//
CASE stCommand.CoordinateType OF
	DUT_Command_CoordinateType.Literal:
		F_AddElement(_Command, _Delimiter, _CoordTypeH);
		F_AddElement(_Command, _Delimiter, LREAL_TO_STRING(stCommand.CoordRef.X));
		F_AddElement(_Command, _Delimiter, LREAL_TO_STRING(stCommand.CoordRef.Y));
		F_AddElement(_Command, _Delimiter, LREAL_TO_STRING(stCommand.CoordRef.Z));
		F_AddElement(_Command, _Delimiter, LREAL_TO_STRING(stCommand.CoordRef.A));
		F_AddElement(_Command, _Delimiter, LREAL_TO_STRING(stCommand.CoordRef.B));
		F_AddElement(_Command, _Delimiter, LREAL_TO_STRING(stCommand.CoordRef.C));
		
	DUT_Command_CoordinateType.Variable:
		F_AddElement(_Command, _Delimiter, _CoordTypeV);
		CASE stCommand.ArrayType OF
			DUT_Command_ArrayType.StoredPosition:
				F_AddElement(_Command, _Delimiter, _ArrayTypeS);
			DUT_Command_ArrayType.VisionRegister:
				F_AddElement(_Command, _Delimiter, _ArrayTypeV);
			DUT_Command_ArrayType.Flag:
				// on damn
		END_CASE
		F_AddElement(_Command, _Delimiter, UDINT_TO_STRING(stCommand.ArrayIndex));
		
END_CASE

// only add if move type is circle
IF stCommand.MoveType = DUT_Command_MoveType.CircularMove THEN
	//
	CASE stCommand.CircleMode OF
		MC_CIRC_MODE.mcCircModeBorder:
			F_AddElement(_Command, _Delimiter, _CircleModeBor);
		MC_CIRC_MODE.mcCircModeCenter:
			F_AddElement(_Command, _Delimiter, _CircleModeCen);
		MC_CIRC_MODE.mcCircModeRadius:
			F_AddElement(_Command, _Delimiter, _CircleModeRad);
	END_CASE
	//
	CASE stCommand.PathChoice OF
		MC_CIRC_PATHCHOICE.mcCircPathChoiceClockwise:
			F_AddElement(_Command, _Delimiter, _PathChoiceClw);
		MC_CIRC_PATHCHOICE.mcCircPathChoiceCounterClockwise:
			F_AddElement(_Command, _Delimiter, _PathChoiceCcw);
	END_CASE
	//
	CASE stCommand.CircularCoordinateType OF
		DUT_Command_CoordinateType.Literal:
			F_AddElement(_Command, _Delimiter, _CoordTypeH);
			F_AddElement(_Command, _Delimiter, LREAL_TO_STRING(stCommand.CoordRef2.X));
			F_AddElement(_Command, _Delimiter, LREAL_TO_STRING(stCommand.CoordRef2.Y));
			F_AddElement(_Command, _Delimiter, LREAL_TO_STRING(stCommand.CoordRef2.Z));
			F_AddElement(_Command, _Delimiter, LREAL_TO_STRING(stCommand.CoordRef2.A));
			F_AddElement(_Command, _Delimiter, LREAL_TO_STRING(stCommand.CoordRef2.B));
			F_AddElement(_Command, _Delimiter, LREAL_TO_STRING(stCommand.CoordRef2.C));
			
		DUT_Command_CoordinateType.Variable:
			F_AddElement(_Command, _Delimiter, _CoordTypeV);
			CASE stCommand.CircularArrayType OF
				DUT_Command_ArrayType.StoredPosition:
					F_AddElement(_Command, _Delimiter, _ArrayTypeS);
				DUT_Command_ArrayType.VisionRegister:
					F_AddElement(_Command, _Delimiter, _ArrayTypeV);
				DUT_Command_ArrayType.Flag:
					// oh damn
			END_CASE
			F_AddElement(_Command, _Delimiter, UDINT_TO_STRING(stCommand.CircularArrayIndex));
			
	END_CASE

END_IF

// set function equal to command
BuildMoveCmd := _Command;

END_FUNCTION

// ---- FB/F_AddElement.TcPOU
FUNCTION F_AddElement
VAR_IN_OUT
	Command: STRING(GVL.COMMAND_LEN);
END_VAR
VAR_INPUT
	Delimiter: STRING(1):=' '; // default to space
	Element: STRING(GVL.COMMAND_LEN);
END_VAR
VAR
END_VAR

//
// input
// 	Element: 'bar'
// 	Delimiter: ','
// 	Command: 'foo'
//
// output
// 	Command: 'foo,bar'
//

Command:=CONCAT(Command, Element);
Command:=CONCAT(Command, Delimiter);

END_FUNCTION

// ---- FB/home/F_HomeOffsetCalc.TcPOU
FUNCTION F_HomeOffsetCalc : LREAL
VAR_INPUT
	CurrentOffset: LREAL;
	CurrentPosition: LREAL;
	HomeSearchDirection: Tc2_MC2.MC_Direction;
END_VAR

IF (HomeSearchDirection = Tc2_MC2.MC_Direction.MC_Negative_Direction) THEN
	F_HomeOffsetCalc := -F_RoundLreal(ABS(CurrentPosition - CurrentOffset),2);
	
ELSIF (HomeSearchDirection = Tc2_MC2.MC_Direction.MC_Positive_Direction) THEN
	F_HomeOffsetCalc := F_RoundLreal(ABS(CurrentPosition - CurrentOffset),2);
	
ELSE
	F_HomeOffsetCalc := CurrentOffset;
	
END_IF

END_FUNCTION

// ---- FB/F_RoundLreal.TcPOU
FUNCTION F_RoundLreal : LREAL
VAR_INPUT
   rIn : LREAL;      
   Digit: INT;         
END_VAR

VAR
   d1 : DINT;
   r0,r1,r2,Rdigit: LREAL;               
END_VAR

// https://forge.codesys.com/forge/talk/Engineering/thread/8d1ee86294/
rdigit   :=INT_TO_LREAL(Digit);
r0 := EXPT(10,rdigit); 
r1 := rIn * r0;
d1 := TRUNC(r1);
r2 := DINT_TO_LREAL(d1);
F_RoundLreal := r2 / r0;

END_FUNCTION

// ---- FB/jog/FB_JogProcessor.TcPOU
FUNCTION_BLOCK FB_JogProcessor
VAR CONSTANT
	NumberOfAxes: UINT:=GVL.NumberOfAxes;
END_VAR
VAR_IN_OUT
	ACS: ARRAY[1..NumberOfAxes] OF AXIS_REF;
	MCS: ARRAY[1..NumberOfAxes] OF AXIS_REF;
	GroupHandler: FB_GroupHandler;
	//Controller: FB_Controller;
END_VAR
VAR_INPUT
	Enable: BOOL;
	Reset: BOOL;
	Velocity: LREAL := 0;
	Acceleration: LREAL := 0;
	Deceleration: LREAL := 0;
	Jerk: LREAL := 0;
    MaxAngularDistance: LREAL := 90.0;
	MaxLinearDistance: LREAL := 50.0;
// 	AccFactor: LREAL := 1.0;
// 	VelFactor: LREAL := 0.1;
// 	JerkFactor: LREAL := 1.0;
// 	TorqueFactor: LREAL := 1.0;
// 	JogForward: ARRAY[1..NumberOfAxes] OF BOOL;
// 	JogBackwards: ARRAY[1..NumberOfAxes] OF BOOL;
	CoordSystem: DUT_CoordSystem := DUT_CoordSystem.TCP;
	ABC_as_ACS: BOOL;
	StoredPositions: REFERENCE TO ARRAY[GVL.POS_ARR_BEG..GVL.POS_ARR_END] OF DUT_StoredPosition;
	VisionRegisters: REFERENCE TO ARRAY[GVL.VIS_ARR_BEG..GVL.VIS_ARR_END] OF DUT_VisionRegister;
	Flags: REFERENCE TO ARRAY[GVL.FLG_ARR_BEG..GVL.FLG_ARR_END] OF DUT_Flags;
END_VAR
VAR_OUTPUT
	Position: DUT_COORD_REF;
	Enabled: BOOL;
	Done: BOOL;
	Busy: BOOL;
	Error: BOOL;
	ErrorID: UDINT;
END_VAR
VAR
	_ResetRtrig: R_TRIG;
	_ErrorRtrig: R_TRIG;
	_EnableRtrig: R_TRIG;
	_EnableFtrig: F_TRIG;
	
	_SequenceMain: INT;
	_SequenceSetCoordTrans: INT;
	
	_MC_Jog: ARRAY[1..NumberOfAxes*2] OF MC_JOG;
	_MC_Halt: ARRAY[1..NumberOfAxes*2] OF MC_HALT;
	_Halt: ARRAY[1..NumberOfAxes*2] OF BOOL;
	_HaltFtrig: ARRAY[1..NumberOfAxes*2] OF F_Trig;
	_JogForward: ARRAY[1..NumberOfAxes] OF BOOL;
	_JogBackwards: ARRAY[1..NumberOfAxes] OF BOOL;
	_CoordSystem: DUT_CoordSystem := DUT_CoordSystem.TCP;
	
	_ControllerCenter: USINT:=128;
	_ControllerDeadZone: USINT:=40;
	
	_OffsetExist: ARRAY[0..GVL.MCS_POS_IDX-GVL.TCP_POS_IDX] OF BOOL;
	
	_MoveToPose: ARRAY[0..GVL.POSE_5_IDX-GVL.POSE_1_IDX] OF BOOL;
	_MoveCommandProcessor: MoveCmdProcessor;
	
	_i, _j, _k: UINT;
	_FirstScan: BOOL:=TRUE;
	
END_VAR

VAR CONSTANT
	STEP_DONE: 				INT := 1000;
	STEP_IDLE: 				INT := 0000;
	STEP_GROUP_ENABLE: 		INT := 0030;
	STEP_WAIT_ENABLE: 		INT := 0035;
	STEP_SET_KINEMATICS: 	INT := 0060;
	STEP_WAIT_KINEMATICS: 	INT := 0070;
	STEP_JOG:				INT := 0080;
	STEP_WAIT_JOG:			INT := 0090;
	STEP_GROUP_DISABLE: 	INT := 0100;
	STEP_WAIT_DISABLE: 		INT := 0110;
END_VAR

_ResetRtrig(CLK:=Reset);

IF _FirstScan THEN
	//
END_IF

//
_M_HandleController();
_M_HandlePose();

//
_EnableFtrig(CLK:=Enable);
IF _EnableFtrig.Q THEN
	//;
END_IF
_EnableRtrig(CLK:=Enable);
IF _EnableRtrig.Q THEN
	//
END_IF

//
CASE _SequenceMain OF
	STEP_DONE: // done
		Busy := FALSE;
		Done := TRUE;
		_SequenceMain := STEP_IDLE;
		
	STEP_IDLE: // IDLE
		IF _EnableRtrig.Q THEN
			Busy := TRUE;
			Done := FALSE;
			_CoordSystem := CoordSystem;
			_M_CheckOffsets();
			_SequenceMain := STEP_GROUP_ENABLE;
		END_IF
		
	STEP_GROUP_ENABLE:
		IF GroupHandler.M_EnableGroup(_CoordSystem) THEN
			_SequenceMain := STEP_WAIT_ENABLE;
		ELSE
			_SequenceMain := STEP_DONE;
			Error := TRUE;
			ErrorID := GroupHandler.ErrorID;
		END_IF
		
	STEP_WAIT_ENABLE:
		// TODO add timeout timer here
		IF GroupHandler.P_GroupReady THEN
			_SequenceMain := STEP_WAIT_JOG;
		END_IF;
		
	STEP_WAIT_JOG: //
		FOR _k:= 1 TO NumberOfAxes DO
			IF _MC_Jog[_k].Error THEN
				Error := TRUE;
				ErrorID := _MC_Jog[_k].ErrorID;
			END_IF
		END_FOR
		IF _EnableFtrig.Q THEN
			_SequenceMain := STEP_GROUP_DISABLE;
			//_SequenceMain := STEP_DONE;
		END_IF
			
	STEP_GROUP_DISABLE:
		IF GroupHandler.M_DisableGroup() THEN
			_SequenceMain := STEP_WAIT_DISABLE;
		ELSE
			_SequenceMain := STEP_DONE;
			Error := TRUE;
			ErrorID := GroupHandler.ErrorID;
		END_IF
		
	STEP_WAIT_DISABLE:
		// TODO add timeouttimer here
		IF NOT GroupHandler.P_GroupReady THEN
			_SequenceMain := STEP_DONE;
		END_IF
	
END_CASE

//
IF _ResetRtrig.Q AND Error THEN
	Error := FALSE;
	ErrorID := 0;
	_SequenceMain := STEP_DONE;
	GroupHandler.M_ResetGroup();
	_MoveCommandProcessor.M_Home();
END_IF

// https://infosys.beckhoff.com/content/1033/tcplclib_tc2_mc2/70120459.html?id=7121036612998147748
FOR _k:= 1 TO NumberOfAxes DO
	_MC_Jog[_k](
		Axis:= ACS[_k], 
		JogForward:= SEL(_CoordSystem = DUT_CoordSystem.ACS, FALSE, _JogForward[_k]), 
		JogBackwards:= SEL(_CoordSystem = DUT_CoordSystem.ACS, FALSE, _JogBackwards[_k]), 
		Mode:= MC_JOGMODE_INCHING, // MC_JOGMODE_STANDARD_SLOW, MC_JOGMODE_STANDARD_FAST, MC_JOGMODE_CONTINUOUS, MC_JOGMODE_INCHING, MC_JOGMODE_INCHING_MODULO
		Position:= MaxAngularDistance, 
		Velocity:= Velocity, 
		Acceleration:= Acceleration, 
		Deceleration:= Deceleration, 
		Jerk:= Jerk, 
		Done=> , 
		Busy=> , 
		Active=> , 
		CommandAborted=> , 
		Error=> , 
		ErrorID=> );
	_MC_Jog[_k+NumberOfAxes](
		Axis:= MCS[_k], 
		JogForward:= SEL(_CoordSystem = DUT_CoordSystem.MCS, FALSE, _JogForward[_k]), 
		JogBackwards:= SEL(_CoordSystem = DUT_CoordSystem.MCS, FALSE, _JogBackwards[_k]), 
		Mode:= MC_JOGMODE_INCHING, // MC_JOGMODE_STANDARD_SLOW, MC_JOGMODE_STANDARD_FAST, MC_JOGMODE_CONTINUOUS, MC_JOGMODE_INCHING, MC_JOGMODE_INCHING_MODULO
		Position:= MaxLinearDistance, 
		Velocity:= Velocity, 
		Acceleration:= Acceleration, 
		Deceleration:= Deceleration, 
		Jerk:= Jerk, 
		Done=> , 
		Busy=> , 
		Active=> , 
		CommandAborted=> , 
		Error=> , 
		ErrorID=> );
END_FOR
FOR _k:= 1 TO NumberOfAxes DO
	IF _MC_Jog[_k].Error OR _MC_Jog[_k+NumberOfAxes].Error THEN
		//
	END_IF
END_FOR

//
FOR _k:= 1 TO NumberOfAxes DO
	_HaltFtrig[_k](CLK:=_JogForward[_k] OR _JogBackwards[_k]);
	IF _HaltFtrig[_k].Q THEN
		_Halt[_k]:=TRUE;
	END_IF
	_HaltFtrig[_k+NumberOfAxes](CLK:=_JogForward[_k] OR _JogBackwards[_k]);
	IF _HaltFtrig[_k+NumberOfAxes].Q THEN
		_Halt[_k+NumberOfAxes]:=TRUE;
	END_IF
END_FOR
FOR _k:= 1 TO NumberOfAxes DO
	_MC_Halt[_k](
		Axis:= ACS[_k], 
		Execute:= _Halt[_k], 
		Deceleration:= Deceleration, 
		Jerk:= Jerk, 
		BufferMode:= , 
		Options:= , 
		Done=> , 
		Busy=> , 
		Active=> , 
		CommandAborted=> , 
		Error=> , 
		ErrorID=> );
	_MC_Halt[_k+NumberOfAxes](
		Axis:= MCS[_k], 
		Execute:= _Halt[_k+NumberOfAxes], 
		Deceleration:= Deceleration, 
		Jerk:= Jerk, 
		BufferMode:= , 
		Options:= , 
		Done=> , 
		Busy=> , 
		Active=> , 
		CommandAborted=> , 
		Error=> , 
		ErrorID=> );
END_FOR
FOR _k:= 1 TO NumberOfAxes DO
	IF _MC_Halt[_k].Done OR _MC_Halt[_k].Error THEN
		_Halt[_k]:=FALSE;
	END_IF
	IF _MC_Halt[_k+NumberOfAxes].Done OR _MC_Halt[_k+NumberOfAxes].Error THEN
		_Halt[_k+NumberOfAxes]:=FALSE;
	END_IF
END_FOR

//
// CoordSystem := _SMC_GroupJog2.CoordSystem;
// ABC_as_ACS := _SMC_GroupJog2.ABC_as_ACS;
// Enabled := _SMC_GroupJog2.Enable;

//
_ErrorRtrig(CLK:=GroupHandler.Error
				//OR _SMC_GroupJog2.Error
				OR _MoveCommandProcessor.Error);			
IF _ErrorRtrig.Q THEN
	// TODO need to rework how error messages are handled (globally)
	// if the move command processor has an error, we dont know what it is.
	Error := TRUE;
END_IF

// do not put anything after this
_FirstScan := FALSE;

METHOD PRIVATE _M_CheckOffsets : BOOL
VAR
	_i: INT;
	_j: INT;
	_k: INT;
END_VAR
IF Enable THEN
	FOR _j:=0 TO GVL.MCS_POS_IDX-GVL.TCP_POS_IDX BY 1 DO
		_OffsetExist[_j] := FALSE;
	END_FOR
	FOR _i := GVL.TCP_POS_IDX TO GVL.MCS_POS_IDX BY 1 DO
		IF StoredPositions[_i].Position.X <> 0
			OR_ELSE StoredPositions[_i].Position.Y <> 0
			OR_ELSE StoredPositions[_i].Position.Z <> 0
			OR_ELSE StoredPositions[_i].Position.A <> 0
			OR_ELSE StoredPositions[_i].Position.B <> 0
			OR_ELSE StoredPositions[_i].Position.C <> 0 THEN
				_OffsetExist[_i - GVL.TCP_POS_IDX] := TRUE;
		END_IF
	END_FOR
END_IF
END_METHOD

METHOD PRIVATE _M_HandleController : BOOL
VAR_STAT
	OptionsTimer: TON := (PT := TIME#1s0ms);
	OptionsRtrig: R_TRIG;
	ShareTimer: TON := (PT := TIME#1s0ms);
	ShareRtrig: R_TRIG;
	OptionsShareRtrig: R_TRIG;
	JogEnabledRtrig: R_TRIG;
	JogEnabledFtrig: F_TRIG;
	SquareButtonRtrig: R_TRIG;
	TriangleButtonRtrig: R_TRIG;
	CircleButtonRtrig: R_TRIG;
	CrossButtonRtrig: R_TRIG;
	R2_Last: USINT;
	JoyStickLeftXLast: USINT;
	JoyStickLeftYLast: USINT;
	JoyStickRightXLast: USINT;
	JoyStickRightYLast: USINT;
	FactorMin: LREAL := 0.01;
END_VAR
// //
// OptionsTimer(IN:=Controller.P_State.Buttons.Options);
// OptionsRtrig(CLK:=Controller.P_State.Buttons.Options);
// //
// ShareTimer(IN:=Controller.P_State.Buttons.Share);
// ShareRtrig(CLK:=Controller.P_State.Buttons.Share);
// //
// OptionsShareRtrig(CLK:=OptionsTimer.Q AND_THEN ShareTimer.Q);
// JogEnabledRtrig(CLK:=Enable);
// JogEnabledFtrig(CLK:=Enable);
// 
// 
// IF Enable AND_THEN Controller.P_State.Connected THEN
// 	
// 	// toggle jog enable
// 	IF OptionsShareRtrig.Q THEN
// 		//_SMC_GroupJog2.Enable := NOT _SMC_GroupJog2.Enable;
// 	END_IF
// 	IF JogEnabledRtrig.Q OR JogEnabledFtrig.Q THEN
// 		IF Enable THEN
// 			_CoordSystem := DUT_CoordSystem.TCP;
// 			Controller.M_SetTriggerMode(E_ControllerTrigger.Right, E_ControllerTriggerMode.Rigid);
// 			Controller.M_SetTriggerForce(E_ControllerTrigger.Right, E_ControllerTriggerForceParameter.One, 0);
// 			Controller.M_SetPlayerID(E_ControllerPlayerID.PlayerALL);
// 			Controller.M_SetMicrophoneState(TRUE);
// 		ELSE
// 			Controller.M_SetTriggerMode(E_ControllerTrigger.Right, E_ControllerTriggerMode.Off);
// 			Controller.M_SetMicrophoneState(FALSE);
// 		END_IF
// 	END_IF
// 	
// 	// cycle through coord system
// 	IF OptionsRtrig.Q AND NOT Controller.P_State.Buttons.Share THEN
// 		CASE _.CoordSystem OF
// 			DUT_CoordSystem.ACS:
// 				_CoordSystem := DUT_CoordSystem.MCS;
// 				Controller.M_SetPlayerID(E_ControllerPlayerID.Player2);
// 			DUT_CoordSystem.MCS:
// 				_CoordSystem := DUT_CoordSystem.UCS1;
// 				Controller.M_SetPlayerID(E_ControllerPlayerID.Player3);
// 			DUT_CoordSystem.UCS1:
// 				_CoordSystem := DUT_CoordSystem.UCS2;
// 				Controller.M_SetPlayerID(E_ControllerPlayerID.Player4);
// 			DUT_CoordSystem.UCS2:
// 				_CoordSystem := DUT_CoordSystem.TCP;
// 				Controller.M_SetPlayerID(E_ControllerPlayerID.PlayerALL);
// 			DUT_CoordSystem.TCP:
// 				_CoordSystem := DUT_CoordSystem.ACS;
// 				Controller.M_SetPlayerID(E_ControllerPlayerID.Player1);
// // 			DUT_CoordSystem.WCS:
// // 				_CoordSystem := DUT_CoordSystem.ACS;
// // 				Controller.M_SetPlayerID(E_ControllerPlayerID.Player1);
// 		END_CASE
// 	END_IF
// 	
// 	// toggle the ABC as ACS setting
// 	IF ShareRtrig.Q AND NOT Controller.P_State.Buttons.Options THEN
// 		ABC_as_ACS := NOT ABC_as_ACS;
// 	END_IF
// 	
// 	// set the velocity factor while the left trigger button is pressed
// 	IF Controller.P_State.Dpad.Left AND_THEN Controller.P_State.Triggers.Right.Two <> R2_Last THEN
// 		R2_Last := Controller.P_State.Triggers.Right.Two;
// 		//_SMC_GroupJog2.VelFactor := MAX(FactorMin, Controller.P_State.Triggers.Right.Two * 1.0 / 255.0);
// 	END_IF
// 	// set the acceleration factor while the up dpad button is pressed
// 	IF Controller.P_State.Dpad.Up AND_THEN Controller.P_State.Triggers.Right.Two <> R2_Last THEN
// 		R2_Last := Controller.P_State.Triggers.Right.Two;
// 		//_SMC_GroupJog2.AccFactor := MAX(FactorMin, Controller.P_State.Triggers.Right.Two * 1.0 / 255.0);
// 	END_IF
// 	// set the jerk factor while the right dpad button is pressed
// 	IF Controller.P_State.Dpad.Right AND_THEN Controller.P_State.Triggers.Right.Two <> R2_Last THEN
// 		R2_Last := Controller.P_State.Triggers.Right.Two;
// 		//_SMC_GroupJog2.JerkFactor := MAX(FactorMin, Controller.P_State.Triggers.Right.Two * 1.0 / 255.0);
// 	END_IF
// 	// set the torque factor while the down dpad down is pressed
// 	IF Controller.P_State.Dpad.Down AND_THEN Controller.P_State.Triggers.Right.Two <> R2_Last THEN
// 		R2_Last := Controller.P_State.Triggers.Right.Two;
// 		//_SMC_GroupJog2.TorqueFactor := MAX(FactorMin, Controller.P_State.Triggers.Right.Two * 1.0 / 255.0);
// 	END_IF
// 	
// 	// first 4 poses can be called using buttons
// 	SquareButtonRtrig(CLK:=Controller.P_State.Buttons.Square);
// 	IF SquareButtonRtrig.Q THEN
// 		M_MoveToPose(E_Pose.One);
// 	END_IF
// 	TriangleButtonRtrig(CLK:=Controller.P_State.Buttons.Triangle);
// 	IF TriangleButtonRtrig.Q THEN
// 		M_MoveToPose(E_Pose.Two);
// 	END_IF
// 	CircleButtonRtrig(CLK:=Controller.P_State.Buttons.Circle);
// 	IF CircleButtonRtrig.Q THEN
// 		M_MoveToPose(E_Pose.Three);
// 	END_IF
// 	CrossButtonRtrig(CLK:=Controller.P_State.Buttons.Cross);
// 	IF CrossButtonRtrig.Q THEN
// 		M_MoveToPose(E_Pose.Four);
// 	END_IF
// 	
// 	//
// 	IF _SequenceMain = STEP_WAIT_JOG THEN
// 		
// 		//
// 		IF Controller.P_State.Joysticks.Left.X <> JoyStickLeftXLast
// 			OR Controller.P_State.Joysticks.Left.Y <> JoyStickLeftYLast THEN
// 				//
// 				JoyStickLeftXLast := Controller.P_State.Joysticks.Left.X;
// 				JoyStickLeftYLast := Controller.P_State.Joysticks.Left.Y;
// 				//	
// 				IF NOT Controller.P_State.Triggers.Left.One THEN
// 					// disable
// 					_JogForward[0] := FALSE;
// 					// disable
// 					_JogBackwards[0] := FALSE;
// 					// Controller.P_State.Joysticks.Left.X // X0-128 is -Y (Backward[1])
// 					_JogBackwards[1] := Controller.P_State.Joysticks.Left.X < _ControllerCenter - _ControllerDeadZone;
// 					// Controller.P_State.Joysticks.Left.X // X128-256 is +Y (Forward[1])
// 					_JogForward[1] := Controller.P_State.Joysticks.Left.X > _ControllerCenter + _ControllerDeadZone;
// 					// Controller.P_State.Joysticks.Left.Y // Y0-128 is +Z (Forward[2])
// 					_JogForward[2] := Controller.P_State.Joysticks.Left.Y < _ControllerCenter - _ControllerDeadZone;
// 					// Controller.P_State.Joysticks.Left.Y // Y128-256 is -Z (Backward[2])
// 					_JogBackwards[2] := Controller.P_State.Joysticks.Left.Y > _ControllerCenter + _ControllerDeadZone;
// 				ELSE
// 					// Controller.P_State.Joysticks.Left.Y // Y0-128 is +X (Forward[0])
// 					_JogForward[0] := Controller.P_State.Joysticks.Left.Y < _ControllerCenter - _ControllerDeadZone;
// 					// Controller.P_State.Joysticks.Left.Y // Y128-256 is -X (Backward[0])
// 					_JogBackwards[0] := Controller.P_State.Joysticks.Left.Y > _ControllerCenter + _ControllerDeadZone;
// 					// disable
// 					_JogBackwards[1] := FALSE;
// 					// disable
// 					_JogForward[1] := FALSE;
// 					// disable
// 					_JogForward[2] := FALSE;
// 					// disable])
// 					_JogBackwards[2] := FALSE;
// 				END_IF
// 		END_IF
// 
// 		//
// 		IF Controller.P_State.Joysticks.Right.X <> JoyStickRightXLast
// 			OR Controller.P_State.Joysticks.Right.Y <> JoyStickRightYLast THEN
// 				//
// 				JoyStickRightXLast := Controller.P_State.Joysticks.Right.X;
// 				JoyStickRightYLast := Controller.P_State.Joysticks.Right.Y;
// 				//				
// 				IF NOT Controller.P_State.Triggers.Right.One THEN
// 					// Controller.P_State.Joysticks.Right.X // X0-128 is +Roll (rot about x) (Forward[3])
// 					_JogBackwards[3] := Controller.P_State.Joysticks.Right.X > _ControllerCenter + _ControllerDeadZone;
// 					// Controller.P_State.Joysticks.Right.X // X128-256 is -Roll (rot about x) (Backward[3])
// 					_JogForward[3] := Controller.P_State.Joysticks.Right.X < _ControllerCenter - _ControllerDeadZone;
// 					// Controller.P_State.Joysticks.Right.Y // Y0-128 is +Pitch (rot about y) (Forward[4])
// 					_JogForward[4] := Controller.P_State.Joysticks.Right.Y < _ControllerCenter - _ControllerDeadZone;
// 					// Controller.P_State.Joysticks.Right.Y // Y128-256 is -Pitch (rot about y) (Backward[4])
// 					_JogBackwards[4] := Controller.P_State.Joysticks.Right.Y > _ControllerCenter + _ControllerDeadZone;
// 					// disable
// 					_JogBackwards[5] := FALSE;
// 					// disable
// 					_JogForward[5] := FALSE;
// 				ELSE
// 					// disable
// 					_JogBackwards[3] := FALSE;
// 					// disable
// 					_JogForward[3] := FALSE;
// 					// disable
// 					_JogForward[4] := FALSE;
// 					// disable
// 					_JogBackwards[4] := FALSE;
// 					// Controller.P_State.Joysticks.Right.X // X0-128 is -Yaw (rot about z) (Backward[5])
// 					_JogBackwards[5] := Controller.P_State.Joysticks.Right.X < _ControllerCenter - _ControllerDeadZone;
// 					// Controller.P_State.Joysticks.Right.X // X128-256 is +Yaw (rot about z) (Forward[5])
// 					_JogForward[5] := Controller.P_State.Joysticks.Right.X > _ControllerCenter + _ControllerDeadZone;
// 				END_IF
// 		END_IF
// 
// 	END_IF
// 	
// END_IF
END_METHOD

METHOD PRIVATE _M_HandlePose : BOOL
VAR
	_MoveCommand: ST_MoveCmd;
	_PoseSpeed: LREAL := 20.0;
	_i, _j, _k: INT;
END_VAR
// FOR _i:=0 TO GVL.POSE_5_IDX - GVL.POSE_1_IDX BY 1 DO
// 	IF _MoveToPose[_i] THEN
// 		_MoveToPose[_i] := FALSE;
// 		//
// 		IF GVL.PowerOn 
// 			AND_THEN PersistentVars.Flags[GVL.HOME_COMPLETE].Value
// 			AND_THEN NOT _MoveCommandProcessor.Busy
// 			AND_THEN NOT _MoveCommandProcessor.Error THEN
// 				//
// 				_MoveCommand.MoveType 			:= DUT_Command_MoveType.DirectMove;
// 				_MoveCommand.PositionType 		:= DUT_Command_PositionType.AbsolutePosition;
// 				_MoveCommand.CoordinateType 	:= DUT_Command_CoordinateType.Literal;
// 				_MoveCommand.Speed 				:= _PoseSpeed;
// 				_MoveCommand.CoordSystem 		:= DUT_CoordSystem.ACS;
// 				_MoveCommand.CoordRef 			:= PersistentVars.StoredPositions[GVL.POSE_1_IDX + _i].Position;
// 				//
// 				_MoveCommandProcessor.Command := BuildMoveCmd(_MoveCommand);
// 				_MoveCommandProcessor.M_Start();
// 				//
// 				EXIT;
// 		END_IF;
// 	END_IF
// END_FOR
// 
// _MoveCommandProcessor(
// 	StoredPositions:= StoredPositions,
// 	VisionRegisters:= VisionRegisters,
// 	Flags:= Flags,
// 	AxisGroup:= AxisGroup, 
// 	GroupHandler:= GroupHandler,
// 	Velocity:= StoredPositions[GVL.SPEEDS_IDX].Position.X, 
// 	VelFactor:= StoredPositions[GVL.SPEEDS_IDX].Position.A,
// 	Acceleration:= StoredPositions[GVL.SPEEDS_IDX].Position.Y, 
// 	AccFactor:= StoredPositions[GVL.SPEEDS_IDX].Position.B,
// 	Jerk:= StoredPositions[GVL.SPEEDS_IDX].Position.Z,
// 	JerkFactor:= StoredPositions[GVL.SPEEDS_IDX].Position.C, 
// 	Position=> ,
// 	ItfUnitMode=> , 
// 	Error=> );
END_METHOD

METHOD M_ClearOffsets : BOOL
VAR
	_i, _j, _k: INT;
END_VAR

FOR _j:=0 TO 3 BY 1 DO
	_OffsetExist[_j] := FALSE;
END_FOR
FOR _i := GVL.TCP_POS_IDX TO GVL.MCS_POS_IDX BY 1 DO
	StoredPositions[_i].Position.X := 0.0;
	StoredPositions[_i].Position.Y := 0.0;
	StoredPositions[_i].Position.Z := 0.0;
	StoredPositions[_i].Position.A := 0.0;
	StoredPositions[_i].Position.B := 0.0;
	StoredPositions[_i].Position.C := 0.0;
END_FOR
END_METHOD

METHOD M_MoveToPose : BOOL
VAR_INPUT
	Pose: E_Pose;
END_VAR
IF Enabled 
	AND NOT _MoveCommandProcessor.Busy
	AND NOT _MoveCommandProcessor.Error THEN
		M_MoveToPose := TRUE;
		_MoveToPose[Pose] := TRUE;
ELSE
	M_MoveToPose := FALSE;
END_IF
END_METHOD

END_FUNCTION_BLOCK

// ---- FB/FB_ProgramProcessor.TcPOU
FUNCTION_BLOCK FB_ProgramProcessor EXTENDS Module
VAR_IN_OUT
	Programs: ARRAY [GVL.PROG_ARR_BEG..GVL.PROG_ARR_END] OF DUT_Program;
	AxisGroup: AXES_GROUP_REF;
	GroupHandler: FB_GroupHandler;
	CmdIO: ST_LogicCmdIO;
END_VAR
VAR_INPUT
	Enable: BOOL;
END_VAR
VAR_OUTPUT
	ItfActiveProcessorUnitMode	: PACK_ML.IUnitMode;
	ItfActiveModule: ItfModule;
	StatusText: STRING(255);
END_VAR
VAR
	_DummyUnitMode: PACK_ML.UnitMode;
	_UnitModeCurrentState: PACK_ML.State;
	_Returning:  ARRAY [GVL.PROG_ARR_BEG..GVL.PROG_ARR_END] OF BOOL;
	_ReturnPrograms: ARRAY [GVL.PROG_ARR_BEG..GVL.PROG_ARR_END] OF UINT;
	_ReturnCommands: ARRAY [GVL.PROG_CMDS_ARR_BEG..GVL.PROG_CMDS_ARR_END + 1] OF UINT; // +1 because we want to be able to tell if calling program was on last command
	_CurrentPrgIdx: UINT;
	_ProcessCommands: FB_CommandProcessor;
	_Commands: ARRAY [GVL.PROG_CMDS_ARR_BEG..GVL.PROG_CMDS_ARR_END] OF DUT_Command;
	_i, _j, _k: INT;
	_FirstScan: BOOL:=TRUE;
END_VAR

VAR CONSTANT
	_STEP_DONE: 			INT := 1000;
	_STEP_IDLE: 			INT := 0000;
	_STEP_PRG:				INT := 0010;
	_STEP_WAIT_EXECUTE:		INT := 0020;
	_STEP_WAIT_IDLE:		INT := 0025;
	_STEP_ERR:              INT := 0030;
END_VAR

//
SUPER^();

//
IF _FirstScan THEN
	// will exception if we don't set this on first scan
	_DummyUnitMode(sName := 'Active Processor', 
					eInitialState := PACK_ML.State.Idle,
					xActive := TRUE);
	ItfActiveProcessorUnitMode := _DummyUnitMode;
END_IF

// this is at best a hack and needs to be rethought out.
// we logically cant assign a process as the active unit mode 
// at start up so we use this dummy one
CASE _DummyUnitMode.CurrentState OF
	PACK_ML.State.Stopped,
	PACK_ML.State.Aborted,
	PACK_ML.State.Held,
	PACK_ML.State.Suspended,
	PACK_ML.State.Complete,
	PACK_ML.State.Idle:
		//
	PACK_ML.State.Resetting,
	PACK_ML.State.Starting,
	PACK_ML.State.Execute,
	PACK_ML.State.Suspending,
	PACK_ML.State.UnSuspending,
	PACK_ML.State.Holding,
	PACK_ML.State.UnHolding,
	PACK_ML.State.Completing,
	PACK_ML.State.Aborting,
	PACK_ML.State.Stopping,
	PACK_ML.State.Clearing:
		_DummyUnitMode.ActingStateCompleted();
END_CASE

// PackML state machine implementation
_UnitModeCurrentState := SUPER^._UnitMode.CurrentState;

//
IF _ProcessCommands.Error THEN
	SUPER^.M_Error(Description:=CONCAT('Command Processor Error: ', _ProcessCommands.ErrorDescription));
	StatusText:=SUPER^.ErrorDescription;
END_IF

//
_ProcessCommands(
	StoredPositions:=SUPER^.StoredPositions,
	VisionRegisters:=SUPER^.VisionRegisters,
	Flags:=SUPER^.Flags,
	AxisGroup:= AxisGroup,
	GroupHandler:= GroupHandler,
	CmdIO:=CmdIO,
	PrgProcessor:= THIS^,
	Enable:= Enable,
	Error=> ,
	StatusText=>StatusText);	

_FirstScan := FALSE;

METHOD PROTECTED M_Aborting : BOOL
CASE _SeqAborting OF
	0:
		_ProcessCommands.M_Abort();
		_SeqAborting := _SeqAborting + 1;
	1:
		IF _ProcessCommands.PropCurrentState = PACK_ML.State.Aborted THEN
			_SeqAborting := 0;
			SUPER^.M_StateComplete();
		END_IF
		
END_CASE

(*IF ItfActiveModule <> 0 THEN
	ItfActiveModule.M_Abort();
	IF ItfActiveModule.PropCurrentState = PACK_ML.State.Aborted THEN
		SUPER^.M_StateComplete();
	END_IF
ELSE
	SUPER^.M_StateComplete();
END_IF*)
END_METHOD

METHOD M_CallProgram : BOOL
VAR_INPUT
	// program to call
	ProgramNumber: UINT;
	// number of the program to return to when the call program ends
	ReturnProgram: UINT;
	// number of the command to start from when called program ends
	ReturnCommand: UINT;
END_VAR
IF ProgramNumber <= GVL.PROG_ARR_END AND_THEN ProgramNumber >= GVL.PROG_ARR_BEG
	AND_THEN ReturnProgram <= GVL.PROG_ARR_END AND_THEN ReturnProgram >= GVL.PROG_ARR_BEG
	AND_THEN SUPER^.PropCurrentState = PACK_ML.State.Execute THEN
		IF _ProcessCommands.M_SetCommands(StartingCommand:=0, Commands:=Programs[ProgramNumber].Commands) THEN
			IF ReturnCommand <= GVL.PROG_CMDS_ARR_END + 1 AND_THEN ReturnCommand >= GVL.PROG_CMDS_ARR_BEG THEN // +1 because we want to be able to tell if calling program was on last command
				_Returning[ProgramNumber] := TRUE;
				_ReturnPrograms[ProgramNumber] := ReturnProgram;
				_ReturnCommands[ProgramNumber] := ReturnCommand;
			END_IF
			_CurrentPrgIdx := ProgramNumber;
			M_CallProgram := TRUE;
		ELSE
			M_CallProgram := FALSE;
		END_IF
ELSE
	M_CallProgram := FALSE;
END_IF
END_METHOD

METHOD PROTECTED M_Clearing : BOOL
SUPER^.M_StateComplete();

(*IF SUPER^.Flags[GVL.HOME_COMPLETE].Value THEN
	CASE _SeqClearing OF
		0:
			_ProcessMoveCommand.M_Home();
			_SeqClearing := _SeqClearing + 1;
		1:
			IF _ProcessMoveCommand.PropCurrentState = PACK_ML.State.Idle THEN
				_SeqClearing := _SeqClearing + 1;
			END_IF
		2:
			IF NOT _ProcessMoveCommand.Error THEN
				_ProcessMoveCommand.Command := GVL.Pose2;
				_ProcessMoveCommand.M_Start();
				_SeqClearing := _SeqClearing + 1;
			ELSE
				SUPER^._M_Error(Description:='Move processor errored. Please reset and try again');
				_SeqClearing := -1;
			END_IF
		3:
			IF _ProcessMoveCommand.PropCurrentState = PACK_ML.State.Execute THEN
				_SeqClearing := _SeqClearing + 1;
			END_IF
		4:
			IF _ProcessMoveCommand.PropCurrentState = PACK_ML.State.Complete 
				OR _ProcessMoveCommand.PropCurrentState = PACK_ML.State.Stopped 
				OR _ProcessMoveCommand.PropCurrentState = PACK_ML.State.Aborted
				OR _ProcessMoveCommand.PropCurrentState = PACK_ML.State.Idle  THEN
					SUPER^.M_StateComplete();
					_SeqClearing := 0;
			END_IF
	END_CASE
ELSE
	SUPER^._M_Error(Description:='Drives are not homed. Please home and try again');
	_SeqClearing := -1;
END_IF

IF _ProcessMoveCommand.Error THEN
	SUPER^._M_Error(Description:='Move processor in error state. Please reset and try again');
	_SeqClearing := -1;
END_IF
*)

(*
IF ItfActiveModule <> 0 THEN
	//
	CASE _Seq OF
		0:
			IF NOT ItfActiveModule.PropCurrentState = PACK_ML.State.Stopped THEN
				ItfActiveModule.M_Abort();
				_Seq := 1;
			ELSE
				SUPER^.M_StateComplete();
			END_IF
		1:
			CASE ItfActiveModule.PropCurrentState OF
				PACK_ML.State.Aborted:
					ItfActiveModule.Clear();
				PACK_ML.State.Stopped:
					_Seq := 0;
			END_CASE
			
	END_CASE
ELSE
	_Seq := 0;
	SUPER^.M_StateComplete();
END_IF
*)
END_METHOD

METHOD PROTECTED M_Complete : BOOL
// once complete, reset to get back to idle
SUPER^._UnitMode.Reset();
END_METHOD

METHOD PROTECTED M_Execute : BOOL
// here we want to execute our commands/jobs/etc and set completed when done.
//
CASE _SeqMain OF
  	_STEP_DONE:
		_SeqMain := _STEP_IDLE;
		
	_STEP_IDLE:
		// hang out here until called to run
		_CurrentPrgIdx := 0;
		SUPER^.M_StateComplete();
		
	_STEP_PRG: //
		IF NOT Enable THEN
			_SeqMain := _STEP_DONE;
		ELSIF _CurrentPrgIdx <= GVL.PROG_ARR_END AND _CurrentPrgIdx >= GVL.PROG_ARR_BEG THEN
			//
			StatusText := '';
			ItfActiveModule := _ProcessCommands;
			ItfActiveProcessorUnitMode := _ProcessCommands.ItfUnitMode;
			
			IF _ProcessCommands.M_SetCommands(StartingCommand:=0, Commands:=Programs[_CurrentPrgIdx].Commands) THEN
				_ProcessCommands.M_Start();
				_SeqMain := _STEP_WAIT_EXECUTE;
			ELSE
				SUPER^.M_Error('Failed to set Command Processor. Check commands.');
				_SeqMain := _STEP_ERR;
			END_IF
			
				
		ELSE
			_SeqMain := _STEP_DONE;
		END_IF
		
	_STEP_WAIT_EXECUTE:
		IF _ProcessCommands.PropCurrentState = PACK_ML.State.Execute THEN
			_SeqMain := _STEP_WAIT_IDLE;
		END_IF
		
	_STEP_WAIT_IDLE: // wait for program to finish
		//
		IF _ProcessCommands.PropCurrentState = PACK_ML.State.Idle THEN
			IF _Returning[_CurrentPrgIdx] THEN
				_Returning[_CurrentPrgIdx] := FALSE;
				IF _ReturnPrograms[_CurrentPrgIdx] <= GVL.PROG_ARR_END AND_THEN _ReturnPrograms[_CurrentPrgIdx] >= GVL.PROG_ARR_BEG
					AND_THEN _ReturnCommands[_CurrentPrgIdx] <= GVL.PROG_CMDS_ARR_END + 1 AND_THEN _ReturnCommands[_CurrentPrgIdx] >= GVL.PROG_CMDS_ARR_BEG // +1 because we want to be able to tell if calling program was on last command
					THEN
						//
						IF _ProcessCommands.M_SetCommands(StartingCommand:=_ReturnCommands[_CurrentPrgIdx], Commands:=Programs[_ReturnPrograms[_CurrentPrgIdx]].Commands) THEN
							_CurrentPrgIdx := _ReturnPrograms[_CurrentPrgIdx];
							_ProcessCommands.M_Start();
							_SeqMain := _STEP_WAIT_EXECUTE;
						ELSE
							SUPER^.M_Error('Failed to set Command Processor. Check commands.');
							_SeqMain := _STEP_ERR;
						END_IF
				ELSE
					_SeqMain := _STEP_DONE;
				END_IF
			ELSE
				_SeqMain := _STEP_DONE;
			END_IF
		END_IF
		//
		IF _ProcessCommands.PropError THEN
			SUPER^._UnitMode.Suspend();
			_SeqMain := _STEP_ERR;
		END_IF
		
	_STEP_ERR: //
	
END_CASE

// watch for rising edge of idle state. this was done for all processors since 
// the vision processor runs in a separate task and isnt guaranteed to start in the same 
// PLC scan.
//_ProcessorDoneRtrig(clk:=ItfActiveProcessorUnitMode.CurrentState = PACK_ML.State.Idle);
END_METHOD

METHOD PROTECTED M_Holding : BOOL
IF ItfActiveModule <> 0 THEN
	ItfActiveModule.M_Hold();
	IF ItfActiveModule.PropCurrentState = PACK_ML.State.Held THEN
		SUPER^.M_StateComplete();
	END_IF
ELSE
	SUPER^.M_StateComplete();
END_IF
END_METHOD

METHOD PROTECTED M_Idle : BOOL
// in this state, we want to reset all the function blocks and hang out
FOR _i:=GVL.PROG_ARR_BEG TO GVL.PROG_ARR_END BY 1 DO
	_Returning[_i] := FALSE;
END_FOR
(*FOR _i:=GVL.PROG_ARR_BEG TO GVL.PROG_ARR_END BY 1 DO
	_ReturnPrograms[_i] := 0;
END_FOR
FOR _i:=GVL.PROG_CMDS_ARR_BEG TO GVL.PROG_CMDS_ARR_END BY 1 DO
	_ReturnCommands[_i] := 0;
END_FOR*)
_SeqMain := _STEP_IDLE;
_SeqAborting := 0;
_SeqClearing := 0;
_SeqResetting := 0;
END_METHOD

METHOD PROTECTED M_Resetting : BOOL
CASE SUPER^._SeqResetting OF
	0:
		_ProcessCommands.M_Home();
		SUPER^._SeqResetting := SUPER^._SeqResetting + 1;
	1:
		IF _ProcessCommands.PropCurrentState = PACK_ML.State.Idle THEN
			SUPER^._SeqResetting := 0;
			SUPER^.M_StateComplete();
		END_IF
		
END_CASE

SUPER^.M_Reset();

(*IF ItfActiveModule <> 0 THEN
	CASE _Seq OF
		0:
			IF NOT ItfActiveModule.PropCurrentState = PACK_ML.State.Idle THEN
				ItfActiveModule.M_Home();
				_Seq := 1;
			ELSE
				SUPER^.M_StateComplete();
			END_IF
		1:
			IF ItfActiveModule.PropCurrentState = PACK_ML.State.Idle THEN
				_Seq := 0;
			END_IF
			
	END_CASE
	
ELSE
	SUPER^.M_StateComplete();
	_Seq := 0;
	
END_IF*)
END_METHOD

METHOD PROTECTED M_SetPackML : BOOL
// SUPER already does this but the default is eInitialState:=PACK_ML.State.Idle 
// and we want PACK_ML.State.Aborted for the Orchestrator
SUPER^._UnitMode(sName := 'Program Processor',
				eInitialState := PACK_ML.State.Aborted,
				xActive := TRUE);
END_METHOD

METHOD M_SetProgram : BOOL
VAR_INPUT
	ProgramNumber: UINT;
END_VAR
IF ProgramNumber >= GVL.PROG_ARR_BEG AND ProgramNumber <= GVL.PROG_ARR_END THEN
	_CurrentPrgIdx := ProgramNumber;
	M_SetProgram := TRUE;
ELSE
	M_SetProgram := FALSE;
END_IF
END_METHOD

METHOD PROTECTED M_Starting : BOOL
// here we want to clear things and get ready for the execute state
// we can consider this the "INIT" state
(*FOR _i:=GVL.PROG_ARR_BEG TO GVL.PROG_ARR_END BY 1 DO
	_Returning[_i] := FALSE;
END_FOR
FOR _i:=GVL.PROG_ARR_BEG TO GVL.PROG_ARR_END BY 1 DO
	_ReturnPrograms[_i] := 0;
END_FOR
FOR _i:=GVL.PROG_CMDS_ARR_BEG TO GVL.PROG_CMDS_ARR_END BY 1 DO
	_ReturnCommands[_i] := 0;
END_FOR*)
//_CurrentPrgIdx := 0;
_SeqMain := _STEP_PRG;
SUPER^.M_StateComplete();
END_METHOD

METHOD PROTECTED M_Stopping : BOOL
IF ItfActiveModule <> 0 THEN
	ItfActiveModule.M_Stop();
	IF ItfActiveModule.PropCurrentState = PACK_ML.State.Idle 
		OR ItfActiveModule.PropCurrentState = PACK_ML.State.Stopped 
		OR ItfActiveModule.PropCurrentState = PACK_ML.State.Aborted 
		OR ItfActiveModule.PropCurrentState = PACK_ML.State.Complete THEN
			SUPER^.M_StateComplete();
	END_IF
	
ELSE
	SUPER^.M_StateComplete();
	
END_IF
END_METHOD

METHOD PROTECTED M_Suspending : BOOL
IF ItfActiveModule <> 0 THEN
	IF ItfActiveModule.PropCurrentState = PACK_ML.State.Execute THEN
		ItfActiveModule.M_Hold();
		IF ItfActiveModule.PropCurrentState = PACK_ML.State.Held THEN
			SUPER^.M_StateComplete();
		END_IF
	ELSE
		SUPER^.M_StateComplete();
	END_IF
	
ELSE
	SUPER^.M_StateComplete();
	
END_IF
END_METHOD

METHOD PROTECTED M_UnHolding : BOOL
//
IF ItfActiveModule <> 0 THEN
	ItfActiveModule.M_Start();
	IF ItfActiveModule.PropCurrentState = PACK_ML.State.Execute THEN
		SUPER^.M_StateComplete();
	END_IF
	
ELSE
	SUPER^.M_StateComplete();
	
END_IF

//
_SeqMain := _STEP_WAIT_IDLE;
END_METHOD

METHOD PROTECTED M_UnSuspending : BOOL
//
IF ItfActiveModule <> 0 THEN
	ItfActiveModule.M_Start();
	IF ItfActiveModule.PropCurrentState = PACK_ML.State.Execute THEN
		SUPER^.M_StateComplete();
	END_IF
	
ELSE
	SUPER^.M_StateComplete();
	
END_IF

//
_SeqMain := _STEP_WAIT_IDLE;
END_METHOD

{attribute 'monitoring' := 'variable'}
PROPERTY P_CurrentCommand : REFERENCE TO DUT_Command
GET
P_CurrentCommand REF= _ProcessCommands.P_CurrentCommand;
END_GET
END_PROPERTY

{attribute 'monitoring' := 'variable'}
PROPERTY P_CurrentCommandIndex : REFERENCE TO UINT
GET
P_CurrentCommandIndex REF= _ProcessCommands.P_CurrentCommandIndex;
END_GET
END_PROPERTY

{attribute 'monitoring' := 'variable'}
PROPERTY P_CurrentProgram : REFERENCE TO UINT
GET
P_CurrentProgram REF= _CurrentPrgIdx;
END_GET
END_PROPERTY

END_FUNCTION_BLOCK

// ---- FB/FB_CommandProcessor.TcPOU
FUNCTION_BLOCK FB_CommandProcessor EXTENDS Module
VAR_IN_OUT
	AxisGroup: AXES_GROUP_REF;
	GroupHandler: FB_GroupHandler;
	CmdIO: ST_LogicCmdIO;
	PrgProcessor: FB_ProgramProcessor;
END_VAR
VAR_INPUT
	Enable: BOOL;
END_VAR
VAR_OUTPUT
	ItfActiveProcessorUnitMode	: PACK_ML.IUnitMode;
	ItfActiveModule: ItfModule;
	StatusText: STRING(255);
END_VAR
VAR
	_Commands: ARRAY [GVL.PROG_CMDS_ARR_BEG..GVL.PROG_CMDS_ARR_END] OF DUT_Command;
	_DummyUnitMode: PACK_ML.UnitMode;
	_UnitModeCurrentState: PACK_ML.State;
	_ActiveCommand: DUT_Command;
	_CurrentCmdIdx: UINT;
	_ProcessMoveCommand: MoveCmdProcessor;
	_ProcessPauseCommand: PauseCmdProcessor;
	_ProcessOutputCommand: OutputCmdProcessor;
	_ProcessorDoneRtrig: R_TRIG;
    //_ProcessVisionCommand: VisionCmdProcessor;
	_ProcessVarSetCommand: VarSetCmdProcessor;
	_ProcessLogicCommand: LogicCmdProcessor;
	_WaitingOnExecute: BOOL;
	_FirstScan: BOOL:=TRUE;
END_VAR

VAR CONSTANT
	_STEP_DONE: 			INT := 1000;
	_STEP_IDLE: 			INT := 0000;
	_STEP_CMD:				INT := 0010;
	_STEP_WAIT:				INT := 0020;
	_STEP_ERR:              INT := 0030;
END_VAR

//
SUPER^();

//
IF _FirstScan THEN
	// will exception if we don't set this on first scan
	_DummyUnitMode(sName := 'Active Processor', 
					eInitialState := PACK_ML.State.Idle,
					xActive := TRUE);
	ItfActiveProcessorUnitMode := _DummyUnitMode;
END_IF

// this is at best a hack and needs to be rethought out.
// we logically cant assign a process as the active unit mode 
// at start up so we use this dummy one
CASE _DummyUnitMode.CurrentState OF
	PACK_ML.State.Stopped,
	PACK_ML.State.Aborted,
	PACK_ML.State.Held,
	PACK_ML.State.Suspended,
	PACK_ML.State.Complete,
	PACK_ML.State.Idle:
		//
	PACK_ML.State.Resetting,
	PACK_ML.State.Starting,
	PACK_ML.State.Execute,
	PACK_ML.State.Suspending,
	PACK_ML.State.UnSuspending,
	PACK_ML.State.Holding,
	PACK_ML.State.UnHolding,
	PACK_ML.State.Completing,
	PACK_ML.State.Aborting,
	PACK_ML.State.Stopping,
	PACK_ML.State.Clearing:
		_DummyUnitMode.ActingStateCompleted();
END_CASE

// PackML state machine implementation
_UnitModeCurrentState := SUPER^._UnitMode.CurrentState;

//
IF _ProcessMoveCommand.Error THEN
	SUPER^.M_Error(Description:=CONCAT('Move Error: ', _ProcessMoveCommand.ErrorDescription));
	StatusText:=SUPER^.ErrorDescription;
END_IF
IF _ProcessPauseCommand.Error THEN
	SUPER^.M_Error(Description:=CONCAT('Pause Error: ', _ProcessPauseCommand.ErrorDescription));
	StatusText:=SUPER^.ErrorDescription;
END_IF
IF _ProcessOutputCommand.Error THEN
	SUPER^.M_Error(Description:=CONCAT('Output Error: ', _ProcessOutputCommand.ErrorDescription));
	StatusText:=SUPER^.ErrorDescription;
END_IF       
// IF _ProcessVisionCommand.Error THEN
// 	SUPER^.M_Error(Description:=CONCAT('Vision Error: ', _ProcessVisionCommand.ErrorDescription));
// 	StatusText:=SUPER^.ErrorDescription;
// END_IF
IF _ProcessVarSetCommand.Error THEN
	SUPER^.M_Error(Description:=CONCAT('Variable Error: ', _ProcessVarSetCommand.ErrorDescription));
	StatusText:=SUPER^.ErrorDescription;
END_IF
IF _ProcessLogicCommand.Error THEN
	SUPER^.M_Error(Description:=CONCAT('Logic Error: ', _ProcessLogicCommand.ErrorDescription));
	StatusText:=SUPER^.ErrorDescription;
END_IF

_ProcessMoveCommand(
	StoredPositions:= SUPER^.StoredPositions,
	VisionRegisters:= SUPER^.VisionRegisters,
	Flags:= SUPER^.Flags,
	AxisGroup:= AxisGroup,
	GroupHandler:= GroupHandler,
	Velocity:= PersistentVars.StoredPositions[GVL.SPEEDS_IDX].Position.X, 
	VelFactor:= PersistentVars.StoredPositions[GVL.SPEEDS_IDX].Position.A,
	Acceleration:= PersistentVars.StoredPositions[GVL.SPEEDS_IDX].Position.Y, 
	AccFactor:= PersistentVars.StoredPositions[GVL.SPEEDS_IDX].Position.B,
	Jerk:= PersistentVars.StoredPositions[GVL.SPEEDS_IDX].Position.Z,
	JerkFactor:= PersistentVars.StoredPositions[GVL.SPEEDS_IDX].Position.C, 
	Position=> ,
	ItfUnitMode=>, 
	Error=> );

_ProcessPauseCommand(
	StoredPositions:= SUPER^.StoredPositions,
	VisionRegisters:= SUPER^.VisionRegisters,
	Flags:= SUPER^.Flags, 
	ElapsedTime=> , 
	RemainingTime=> , 
	ItfUnitMode=>, 
	Error=> );

_ProcessOutputCommand(
	StoredPositions:= SUPER^.StoredPositions,
	VisionRegisters:= SUPER^.VisionRegisters,
	Flags:= SUPER^.Flags,
	Digital:= CmdIO.Output,
	Pwm:= CmdIO.Pwm,
	Enable:= Enable,
	ItfUnitMode=>, 
	Error=> );
	
_ProcessVarSetCommand( 
	StoredPositions:= SUPER^.StoredPositions,
	VisionRegisters:= SUPER^.VisionRegisters,
	Flags:= SUPER^.Flags,
	ItfUnitMode=>, 
	Error=> , 
	ErrorDescription=> );
	
_ProcessLogicCommand(
	StoredPositions:= SUPER^.StoredPositions,
	VisionRegisters:= SUPER^.VisionRegisters,
	Flags:= SUPER^.Flags,
	CmdProcessor:= THIS^,
	PrgProcessor:= PrgProcessor,
	ItfUnitMode=>, 
	Error=> , 
	ErrorDescription=> , 
	CmdIO:= CmdIO);

// _ProcessVisionCommand(
// 	VisionSystemIpAddress:= PersistentVars.VisionSystemIpAddress,
// 	VisionSystemPort:= PersistentVars.VisionSystemPort,
// 	StoredPositions:= PersistentVars.StoredPositions,
// 	VisionRegisters:= PersistentVars.VisionRegisters,
// 	Flags:= PersistentVars.Flags,
// 	LogicCmdIO:= CmdIO,
// 	ItfUnitMode=> ,
// 	Error=> , 
// 	ErrorDescription=> , 
// 	VisionStateText=> );
	
_FirstScan := FALSE;

METHOD PROTECTED M_Aborting : BOOL
CASE _SeqAborting OF
	0:
		_ProcessMoveCommand.M_Abort();
		_ProcessPauseCommand.M_Abort();
		_ProcessOutputCommand.M_Abort();
// 		_ProcessVisionCommand.M_Abort();
		_ProcessVarSetCommand.M_Abort();
		_ProcessLogicCommand.M_Abort();
		_SeqAborting := _SeqAborting + 1;
	1:
		IF _ProcessMoveCommand.PropCurrentState = PACK_ML.State.Aborted
			AND _ProcessPauseCommand.PropCurrentState = PACK_ML.State.Aborted 
			//AND _ProcessInputCommand.PropCurrentState = PACK_ML.State.Aborted
			AND _ProcessOutputCommand.PropCurrentState = PACK_ML.State.Aborted
			//AND _ProcessVisionCommand.PropCurrentState = PACK_ML.State.Aborted
			AND _ProcessVarSetCommand.PropCurrentState = PACK_ML.State.Aborted
			AND _ProcessLogicCommand.PropCurrentState = PACK_ML.State.Aborted THEN
				_SeqAborting := 0;
				SUPER^.M_StateComplete();
		END_IF
		
END_CASE

(*IF ItfActiveModule <> 0 THEN
	ItfActiveModule.M_Abort();
	IF ItfActiveModule.PropCurrentState = PACK_ML.State.Aborted THEN
		SUPER^.M_StateComplete();
	END_IF
ELSE
	SUPER^.M_StateComplete();
END_IF*)
END_METHOD

METHOD PROTECTED M_Clearing : BOOL
SUPER^.M_StateComplete();

(*IF SUPER^.Flags[GVL.HOME_COMPLETE].Value THEN
	CASE _SeqClearing OF
		0:
			_ProcessMoveCommand.M_Home();
			_SeqClearing := _SeqClearing + 1;
		1:
			IF _ProcessMoveCommand.PropCurrentState = PACK_ML.State.Idle THEN
				_SeqClearing := _SeqClearing + 1;
			END_IF
		2:
			IF NOT _ProcessMoveCommand.Error THEN
				_ProcessMoveCommand.Command := GVL.Pose2;
				_ProcessMoveCommand.M_Start();
				_SeqClearing := _SeqClearing + 1;
			ELSE
				SUPER^._M_Error(Description:='Move processor errored. Please reset and try again');
				_SeqClearing := -1;
			END_IF
		3:
			IF _ProcessMoveCommand.PropCurrentState = PACK_ML.State.Execute THEN
				_SeqClearing := _SeqClearing + 1;
			END_IF
		4:
			IF _ProcessMoveCommand.PropCurrentState = PACK_ML.State.Complete 
				OR _ProcessMoveCommand.PropCurrentState = PACK_ML.State.Stopped 
				OR _ProcessMoveCommand.PropCurrentState = PACK_ML.State.Aborted
				OR _ProcessMoveCommand.PropCurrentState = PACK_ML.State.Idle  THEN
					SUPER^.M_StateComplete();
					_SeqClearing := 0;
			END_IF
	END_CASE
ELSE
	SUPER^._M_Error(Description:='Drives are not homed. Please home and try again');
	_SeqClearing := -1;
END_IF

IF _ProcessMoveCommand.Error THEN
	SUPER^._M_Error(Description:='Move processor in error state. Please reset and try again');
	_SeqClearing := -1;
END_IF
*)

(*
IF ItfActiveModule <> 0 THEN
	//
	CASE _Seq OF
		0:
			IF NOT ItfActiveModule.PropCurrentState = PACK_ML.State.Stopped THEN
				ItfActiveModule.M_Abort();
				_Seq := 1;
			ELSE
				SUPER^.M_StateComplete();
			END_IF
		1:
			CASE ItfActiveModule.PropCurrentState OF
				PACK_ML.State.Aborted:
					ItfActiveModule.Clear();
				PACK_ML.State.Stopped:
					_Seq := 0;
			END_CASE
			
	END_CASE
ELSE
	_Seq := 0;
	SUPER^.M_StateComplete();
END_IF
*)
END_METHOD

METHOD PROTECTED M_Complete : BOOL
// once complete, reset to get back to idle
SUPER^._UnitMode.Reset();
END_METHOD

METHOD PROTECTED M_Execute : BOOL
// here we want to execute our commands/jobs/etc and set completed when done.
//
CASE _SeqMain OF
  	_STEP_DONE:
		_SeqMain := _STEP_IDLE;
		
	_STEP_IDLE:
		// hang out here until called to run
		_WaitingOnExecute := FALSE;
		_CurrentCmdIdx := 0;
		SUPER^.M_StateComplete();
		
	_STEP_CMD: //
		IF NOT Enable THEN
			_SeqMain := _STEP_DONE;
			
		ELSIF _CurrentCmdIdx <= GVL.PROG_CMDS_ARR_END AND _CurrentCmdIdx >= GVL.PROG_CMDS_ARR_BEG THEN
			//
			IF _Commands[_CurrentCmdIdx].CommandType = DUT_CommandType.Disabled THEN
				// want to increment here so that we can disable some commands 
				// in the program and it continue to execute
				_CurrentCmdIdx := _CurrentCmdIdx + 1;
				_SeqMain := _STEP_CMD;
				
			ELSE
				IF NOT _WaitingOnExecute THEN
					CASE _Commands[_CurrentCmdIdx].CommandType OF
						DUT_CommandType.MoveCommand: //
							StatusText := 'Move Command in Progress.';
							ItfActiveProcessorUnitMode := _ProcessMoveCommand.ItfUnitMode;
							ItfActiveModule := _ProcessMoveCommand;
							_ProcessMoveCommand.Command := _Commands[_CurrentCmdIdx].CommandString;
							ItfActiveModule.M_Start();
							_WaitingOnExecute := TRUE;
						
						DUT_CommandType.PauseCommand: //
							StatusText := 'Pause Command in Progress.';
							ItfActiveProcessorUnitMode := _ProcessPauseCommand.ItfUnitMode;
							ItfActiveModule := _ProcessPauseCommand;
							_ProcessPauseCommand.Command := _Commands[_CurrentCmdIdx].CommandString;
							ItfActiveModule.M_Start();
							_WaitingOnExecute := TRUE;
						
						DUT_CommandType.OutputCommand: //
							StatusText := 'Output Command in Progress.';
							ItfActiveProcessorUnitMode := _ProcessOutputCommand.ItfUnitMode;
							ItfActiveModule := _ProcessOutputCommand;
							_ProcessOutputCommand.Command := _Commands[_CurrentCmdIdx].CommandString;
							ItfActiveModule.M_Start();
							_WaitingOnExecute := TRUE;
						
	// 					DUT_CommandType.VisionCommand: //
	// 						StatusText := 'Vision Command in Progress.';
	// 						ItfActiveProcessorUnitMode := _ProcessVisionCommand.ItfUnitMode;
	// 						ItfActiveModule := _ProcessVisionCommand;
	// 						_ProcessVisionCommand.Command := _Commands[_CurrentCmdIdx].CommandString;
	// 						ItfActiveModule.M_Start();
	//						_WaitingOnExecute := TRUE;
						
						DUT_CommandType.VarSetCommand: //
							StatusText := 'VarSet Command in Progress.';
							ItfActiveProcessorUnitMode := _ProcessVarsetCommand.ItfUnitMode;
							ItfActiveModule := _ProcessVarsetCommand;
							_ProcessVarsetCommand.Command := _Commands[_CurrentCmdIdx].CommandString;
							ItfActiveModule.M_Start();
							_WaitingOnExecute := TRUE;
						
						DUT_CommandType.LogicCommand: //
							StatusText := 'Logic Command in Progress.';
							ItfActiveProcessorUnitMode := _ProcessLogicCommand.ItfUnitMode;
							ItfActiveModule := _ProcessLogicCommand;
							_ProcessLogicCommand.Command := _Commands[_CurrentCmdIdx].CommandString;
							ItfActiveModule.M_Start();
							_WaitingOnExecute := TRUE;
							
					ELSE
						_SeqMain := _STEP_CMD;
						
					END_CASE
				END_IF
				
				// wait for executing
				IF ItfActiveModule.PropCurrentState = PACK_ML.State.Execute THEN
					_WaitingOnExecute := FALSE;
					_ActiveCommand := _Commands[_CurrentCmdIdx];
					_CurrentCmdIdx := _CurrentCmdIdx + 1;
					_SeqMain := _STEP_WAIT;
				END_IF
			END_IF
				
		ELSE
			_SeqMain := _STEP_DONE;
		END_IF
		
	_STEP_WAIT: // wait for command to finish
		//
		IF _ProcessorDoneRtrig.Q THEN
			_SeqMain := _STEP_CMD;
		END_IF
		//
		IF ItfActiveModule.PropError THEN
			SUPER^._UnitMode.Suspend();
			_SeqMain := _STEP_ERR;
		END_IF
		
	_STEP_ERR: //
	
END_CASE

// watch for rising edge of idle state. this was done for all processors since 
// the vision processor runs in a separate task and isnt guaranteed to start in the same 
// PLC scan.
_ProcessorDoneRtrig(clk:=ItfActiveProcessorUnitMode.CurrentState = PACK_ML.State.Idle);
END_METHOD

METHOD PROTECTED M_Holding : BOOL
IF ItfActiveModule <> 0 THEN
	ItfActiveModule.M_Hold();
	IF ItfActiveModule.PropCurrentState = PACK_ML.State.Held THEN
		SUPER^.M_StateComplete();
	END_IF
ELSE
	SUPER^.M_StateComplete();
END_IF
END_METHOD

METHOD PROTECTED M_Idle : BOOL
// in this state, we want to reset all the function blocks and hang out
_SeqMain := _STEP_IDLE;
_SeqAborting := 0;
_SeqClearing := 0;
_SeqResetting := 0;
END_METHOD

METHOD PROTECTED M_Resetting : BOOL
CASE SUPER^._SeqResetting OF
	0:
		_ProcessMoveCommand.M_Home();
		_ProcessPauseCommand.M_Home();
		//_ProcessInputCommand.M_Home();
		_ProcessOutputCommand.M_Home();
		//_ProcessVisionCommand.M_Home();
		_ProcessVarSetCommand.M_Home();
		_ProcessLogicCommand.M_Home();
		SUPER^._SeqResetting := SUPER^._SeqResetting + 1;
	1:
		IF _ProcessMoveCommand.PropCurrentState = PACK_ML.State.Idle
			AND _ProcessPauseCommand.PropCurrentState = PACK_ML.State.Idle 
			AND _ProcessOutputCommand.PropCurrentState = PACK_ML.State.Idle
			//AND _ProcessVisionCommand.PropCurrentState = PACK_ML.State.Idle
			AND _ProcessVarSetCommand.PropCurrentState = PACK_ML.State.Idle
			AND _ProcessLogicCommand.PropCurrentState = PACK_ML.State.Idle THEN
				SUPER^._SeqResetting := 0;
				SUPER^.M_StateComplete();
		END_IF
		
END_CASE

SUPER^.M_Reset();

(*IF ItfActiveModule <> 0 THEN
	CASE _Seq OF
		0:
			IF NOT ItfActiveModule.PropCurrentState = PACK_ML.State.Idle THEN
				ItfActiveModule.M_Home();
				_Seq := 1;
			ELSE
				SUPER^.M_StateComplete();
			END_IF
		1:
			IF ItfActiveModule.PropCurrentState = PACK_ML.State.Idle THEN
				_Seq := 0;
			END_IF
			
	END_CASE
	
ELSE
	SUPER^.M_StateComplete();
	_Seq := 0;
	
END_IF*)
END_METHOD

METHOD M_SetCommands : BOOL
VAR_INPUT
	StartingCommand: UINT;
	Commands: ARRAY[GVL.PROG_CMDS_ARR_BEG..GVL.PROG_CMDS_ARR_END] OF DUT_Command;
END_VAR
IF StartingCommand >= GVL.PROG_CMDS_ARR_BEG AND StartingCommand <= GVL.PROG_CMDS_ARR_END + 1 THEN // +1 because we want to be able to tell if calling program was on last command
	_CurrentCmdIdx := StartingCommand;
	_Commands := Commands;
	M_SetCommands := TRUE;
ELSE
	M_SetCommands := FALSE;
END_IF
END_METHOD

METHOD M_SetNextCommand : BOOL
VAR_INPUT
	CommandNumber: UINT;
END_VAR
IF CommandNumber <= GVL.PROG_CMDS_ARR_END AND CommandNumber >= GVL.PROG_CMDS_ARR_BEG THEN
	_CurrentCmdIdx := CommandNumber;
	M_SetNextCommand := TRUE;
ELSE
	M_SetNextCommand := FALSE;
END_IF
END_METHOD

METHOD PROTECTED M_SetPackML : BOOL
// SUPER already does this but the default is eInitialState:=PACK_ML.State.Idle 
// and we want PACK_ML.State.Aborted for the Orchestrator
SUPER^._UnitMode(sName := 'Command Processor',
				eInitialState := PACK_ML.State.Aborted,
				xActive := TRUE);
END_METHOD

METHOD PROTECTED M_Starting : BOOL
// here we want to clear things and get ready for the execute state
// we can consider this the "INIT" state
_SeqMain := _STEP_CMD;
SUPER^._TimeoutTimer.PT := T#0MS; // timeout is ignored if set to 0
SUPER^.M_StateComplete();
END_METHOD

METHOD PROTECTED M_Stopping : BOOL
IF ItfActiveModule <> 0 THEN
	ItfActiveModule.M_Stop();
	IF ItfActiveModule.PropCurrentState = PACK_ML.State.Idle 
		OR ItfActiveModule.PropCurrentState = PACK_ML.State.Stopped 
		OR ItfActiveModule.PropCurrentState = PACK_ML.State.Aborted 
		OR ItfActiveModule.PropCurrentState = PACK_ML.State.Complete THEN
			SUPER^.M_StateComplete();
	END_IF
	
ELSE
	SUPER^.M_StateComplete();
	
END_IF
END_METHOD

METHOD PROTECTED M_Suspending : BOOL
IF ItfActiveModule <> 0 THEN
	IF ItfActiveModule.PropCurrentState = PACK_ML.State.Execute THEN
		ItfActiveModule.M_Hold();
		IF ItfActiveModule.PropCurrentState = PACK_ML.State.Held THEN
			SUPER^.M_StateComplete();
		END_IF
	ELSE
		SUPER^.M_StateComplete();
	END_IF
	
ELSE
	SUPER^.M_StateComplete();
	
END_IF
END_METHOD

METHOD PROTECTED M_UnHolding : BOOL
//
IF ItfActiveModule <> 0 THEN
	ItfActiveModule.M_Start();
	IF ItfActiveModule.PropCurrentState = PACK_ML.State.Execute THEN
		SUPER^.M_StateComplete();
	END_IF
	
ELSE
	SUPER^.M_StateComplete();
	
END_IF

//
_SeqMain := _STEP_WAIT;
END_METHOD

METHOD PROTECTED M_UnSuspending : BOOL
//
IF ItfActiveModule <> 0 THEN
	ItfActiveModule.M_Start();
	IF ItfActiveModule.PropCurrentState = PACK_ML.State.Execute THEN
		SUPER^.M_StateComplete();
	END_IF
	
ELSE
	SUPER^.M_StateComplete();
	
END_IF

//
_SeqMain := _STEP_WAIT;
END_METHOD

{attribute 'monitoring' := 'variable'}
PROPERTY P_CurrentCommand : REFERENCE TO DUT_Command
GET
P_CurrentCommand REF= _ActiveCommand;
END_GET
END_PROPERTY

{attribute 'monitoring' := 'variable'}
PROPERTY P_CurrentCommandIndex : REFERENCE TO UINT
GET
P_CurrentCommandIndex REF= _CurrentCmdIdx;
END_GET
END_PROPERTY

END_FUNCTION_BLOCK

// ---- FB/pause/PauseCmdProcessor.TcPOU
FUNCTION_BLOCK PauseCmdProcessor EXTENDS Module
VAR_INPUT
	Command: STRING(GVL.COMMAND_LEN):='';
END_VAR
VAR_OUTPUT
	ElapsedTime: TIME;
	RemainingTime: TIME;
END_VAR
VAR
	_Timer: TON;
	_Timer_IN: BOOL;
	_Timer_PT: TIME;
	_Timer_Q: BOOL;
	_Timer_ET: TIME;
END_VAR
VAR
	_UnitModeCurrentState: PACK_ML.State;
	_ParsePauseCmd: ParsePauseCmd;
END_VAR
VAR CONSTANT
	_STEP_DONE: 		INT := 1000;
	_STEP_IDLE: 		INT := 0000;
	_STEP_COMMAND: 		INT := 0010;
	_STEP_TWO: 			INT := 0020;
	_STEP_ERR: 			INT := 0030;
END_VAR

SUPER^();

// PackML state machine implementation
_UnitModeCurrentState := SUPER^._UnitMode.CurrentState;

//
CASE SUPER^._SeqMain OF
	
    _STEP_DONE:
 		_Timer_IN := FALSE;
		SUPER^._SeqMain := _STEP_IDLE;
        
    _STEP_IDLE:
		// hang out here until called to run
        
    _STEP_COMMAND:
		_ParsePauseCmd(Command:=Command);
		_Timer_PT := _ParsePauseCmd.stCommand.PauseTime;
 		_Timer_IN := TRUE;
		// next, please
		SUPER^._SeqMain := _STEP_TWO;
		
	_STEP_TWO:
		IF _Timer.Q THEN
			// next, please
			SUPER^._SeqMain := _STEP_DONE;
		END_IF

END_CASE

_Timer(
	IN:= _Timer_IN, 
	PT:= _Timer_PT, 
	Q=> _Timer_Q, 
	ET=> _Timer_ET);
	
ElapsedTime := _Timer_ET;
RemainingTime := _Timer_PT - _Timer_ET;

METHOD PROTECTED M_Complete : BOOL
// once complete, reset to get back to idle
SUPER^._UnitMode.Reset();
END_METHOD

METHOD PROTECTED M_Execute : BOOL
// here we want to execute our commands/jobs/etc and set completed when done.
IF SUPER^._SeqMain =_STEP_IDLE THEN
	SUPER^.M_StateComplete();
END_IF
END_METHOD

METHOD PROTECTED M_Resetting : BOOL
CASE SUPER^._SeqResetting OF
	0:
		_Timer_IN := FALSE;
		_SeqResetting := _SeqResetting + 1;
	1:
		IF NOT _Timer_IN THEN
			SUPER^.M_StateComplete();
			_SeqResetting := 0;
		END_IF
END_CASE
END_METHOD

METHOD PROTECTED M_SetPackML : BOOL
SUPER^._UnitMode(	sName := 'Pause Processor',
				eInitialState := PACK_ML.State.Idle,
				xActive := TRUE);
END_METHOD

METHOD PROTECTED M_Starting : BOOL
// here we want to clear things and get ready for the execute state
// I can consider this the "INIT" state
SUPER^._SeqMain := _STEP_COMMAND;
SUPER^.M_StateComplete();
END_METHOD

END_FUNCTION_BLOCK

// ---- FB/pause/ParsePauseCmd.TcPOU
FUNCTION_BLOCK ParsePauseCmd
VAR_INPUT
	Command: STRING(GVL.COMMAND_LEN);
END_VAR
VAR_OUTPUT
	stCommand: ST_PauseCmd;
	Error: BOOL;
	ErrorDescription: STRING;
END_VAR
VAR
	_CmdParams: ARRAY [0..GVL.COMMAND_LEN] OF STRING;
END_VAR

// T#30s

Error:=FALSE;
ErrorDescription:='';

// split command string into commands
_CmdParams:=F_SplitCmd(Command:=Command);

stCommand.PauseTime := STRING_TO_TIME(_CmdParams[0]);

END_FUNCTION_BLOCK

// ---- FB/output/OutputCmdProcessor.TcPOU
FUNCTION_BLOCK OutputCmdProcessor EXTENDS Module
VAR_INPUT
	Enable: BOOL;
	Command: STRING(GVL.COMMAND_LEN):='';
END_VAR
VAR_IN_OUT
	Digital: ARRAY [GVL.DIG_OUT_ARR_BEG..GVL.DIG_OUT_ARR_END] OF BOOL;
	Pwm: ARRAY [GVL.PWM_OUT_ARR_BEG..GVL.PWM_OUT_ARR_END] OF BYTE;
END_VAR
VAR_OUTPUT
END_VAR
VAR
END_VAR
VAR
	_RunRtrig: R_TRIG;
	_SequenceDigital: INT;
	_SequencePwm: INT;
	
	_UnitModeCurrentState: PACK_ML.State;
	_OutputCommandParser: ParseOutputCmd;
	_OutputType: DUT_OutputType;
	_OutputTarget: INT;
	_OutputValue1: LREAL;
END_VAR
VAR CONSTANT
	_STEP_DONE: 		INT := 1000;
	_STEP_IDLE: 		INT := 0000;
	_STEP_COMMAND: 		INT := 0010;
	_STEP_TWO: 			INT := 0020;
	_STEP_ERR: 			INT := 0030;
END_VAR

SUPER^();

// PackML state machine implementation
_UnitModeCurrentState := SUPER^._UnitMode.CurrentState;

//
CASE SUPER^._SeqMain OF
	
    _STEP_DONE:
		SUPER^._SeqMain := _STEP_IDLE;
        
    _STEP_IDLE:
        // hang out here untill called to run
		
    _STEP_COMMAND:
		_OutputCommandParser(Command:=Command);
		IF _OutputCommandParser.Error THEN
			SUPER^.M_Error(Description:=_OutputCommandParser.ErrorDescription);
			SUPER^._SeqMain := _STEP_ERR;
		ELSE
			_OutputType := _OutputCommandParser.stCommand.OutputType;
			_OutputTarget := _OutputCommandParser.stCommand.OutputTarget;
			_OutputValue1 := _OutputCommandParser.stCommand.OutputValue1;
			
			CASE _OutputType OF
				DUT_OutputType.Digital: //
					_SequenceDigital := 1;
					SUPER^._SeqMain := _STEP_TWO;
				DUT_OutputType.Pwm: //
					_SequencePwm := 1;
					SUPER^._SeqMain := _STEP_TWO;
			ELSE
				SUPER^._SeqMain := _STEP_DONE;
				
			END_CASE
		END_IF
		
	_STEP_TWO:
		IF _SequenceDigital = 0 
			AND _SequencePwm = 0 THEN
				// next, please
				SUPER^._SeqMain := _STEP_DONE;
		END_IF;

END_CASE

CASE _SequenceDigital OF
	0: //
	1: //
		THIS^.Digital[_OutputTarget] := _OutputValue1 > 0;
		_SequenceDigital := 0;
END_CASE

CASE _SequencePwm OF
	0: //
	1: //
		THIS^.Pwm[_OutputTarget] := LREAL_TO_BYTE(_OutputValue1);
		_SequencePwm := 0;
	
END_CASE

METHOD PROTECTED M_Aborting : BOOL
CASE SUPER^._SeqAborting OF
	0:
		SUPER^._SeqAborting := SUPER^._SeqAborting + 1;
	1:
		SUPER^.M_StateComplete();
		SUPER^._SeqAborting := 0;
		
END_CASE
END_METHOD

METHOD PROTECTED M_Clearing : BOOL
_SequenceDigital := 0;
_SequencePwm := 0;

SUPER^.M_StateComplete();
END_METHOD

METHOD PROTECTED M_Complete : BOOL
// once complete, reset to get back to idle
SUPER^._UnitMode.Reset();
END_METHOD

METHOD PROTECTED M_Execute : BOOL
// here we want to execute our commands/jobs/etc and set completed when done.
IF SUPER^._SeqMain =_STEP_IDLE THEN
	SUPER^.M_StateComplete();
END_IF
END_METHOD

METHOD PROTECTED M_Holding : BOOL
CASE SUPER^._SeqHolding OF
	0:
		SUPER^._SeqHolding := SUPER^._SeqHolding + 1;
	1:
		SUPER^.M_StateComplete();
		SUPER^._SeqHolding := 0;
		
END_CASE
END_METHOD

METHOD PROTECTED M_Idle : BOOL
_SequenceDigital := 0;
_SequencePwm := 0;
SUPER^._SeqMain := 0;
END_METHOD

METHOD PROTECTED M_Resetting : BOOL
CASE SUPER^._SeqResetting OF
	0:
		_SeqResetting := _SeqResetting + 1;
	1:
		SUPER^.M_StateComplete();
		_SeqResetting := 0;
END_CASE
END_METHOD

METHOD PROTECTED M_SetPackML : BOOL
SUPER^._UnitMode(	sName := 'Output Processor',
				eInitialState := PACK_ML.State.Idle,
				xActive := TRUE);
END_METHOD

METHOD PROTECTED M_Starting : BOOL
// here we want to clear things and get ready for the execute state
// I can consider this the "INIT" state
SUPER^._SeqMain := _STEP_COMMAND;
SUPER^.M_StateComplete();
END_METHOD

METHOD PROTECTED M_UnHolding : BOOL

//
SUPER^._SeqMain := _STEP_COMMAND;

//
SUPER^.M_StateComplete();
END_METHOD

END_FUNCTION_BLOCK

// ---- FB/output/ParseOutputCmd.TcPOU
FUNCTION_BLOCK ParseOutputCmd
VAR_INPUT
	Command: STRING(GVL.COMMAND_LEN);
END_VAR
VAR_OUTPUT
	stCommand: ST_OutputCmd;
	Error: BOOL;
	ErrorDescription: STRING;
END_VAR
VAR
	_CmdParams: ARRAY [0..GVL.COMMAND_LEN] OF STRING;
	_OutputType: STRING;
END_VAR

// DIG +0001.00 +0001.00 (turn digital input 1 on)
// DIG +0001.00 +0000.00 (turn digital input 1 off)
// PWM +0001.00 +0030.00(set PWM 1 to position 30)

Error:=FALSE;
ErrorDescription:='';

// split command string into commands
_CmdParams:=F_SplitCmd(Command:=Command);

_OutputType := _CmdParams[0];
IF _OutputType = 'DIG' THEN
	stCommand.OutputType := DUT_OutputType.Digital;
ELSIF _OutputType = 'PWM' THEN
	stCommand.OutputType := DUT_OutputType.Pwm;
END_IF
stCommand.OutputTarget := STRING_TO_INT(_CmdParams[1]);
stCommand.OutputValue1 := STRING_TO_LREAL(_CmdParams[2]);

END_FUNCTION_BLOCK

// ---- FB/varset/VarSetCmdProcessor.TcPOU
FUNCTION_BLOCK VarSetCmdProcessor EXTENDS Module
VAR_INPUT
	Command: STRING(GVL.COMMAND_LEN):='';
END_VAR
VAR_OUTPUT
END_VAR
VAR
END_VAR
VAR CONSTANT
	_STEP_DONE: 		INT := 1000;
	_STEP_IDLE: 		INT := 0000;
	_STEP_COMMAND: 		INT := 0010;
	_STEP_ERR: 			INT := 0020;
END_VAR
VAR
	_UnitModeCurrentState: PACK_ML.State;
	_VarSetCmdParser: ParseVarSetCmd;
END_VAR

SUPER^();

// PackML state machine implementation
_UnitModeCurrentState := SUPER^._UnitMode.CurrentState;

//
CASE SUPER^._SeqMain OF
    _STEP_DONE:
		SUPER^._SeqMain := _STEP_IDLE;
        
    _STEP_IDLE:
		// hang out here until called to run
		
	_STEP_COMMAND:
        _VarSetCmdParser(Command:=Command);
		IF _VarSetCmdParser.Error THEN
			//
			SUPER^.M_Error(Description:=_VarSetCmdParser.ErrorDescription);
			// next, please
			SUPER^._SeqMain := _STEP_ERR;
			
		ELSE
			//
			IF _VarSetCmdParser.stCommand.ArrayType = DUT_Command_ArrayType.StoredPosition THEN
				SUPER^.StoredPositions[_VarSetCmdParser.stCommand.ArrayIndex].Position := _VarSetCmdParser.stCommand.Coordinates;
			ELSIF _VarSetCmdParser.stCommand.ArrayType = DUT_Command_ArrayType.VisionRegister THEN
				SUPER^.VisionRegisters[_VarSetCmdParser.stCommand.ArrayIndex].Position := _VarSetCmdParser.stCommand.Coordinates;
			ELSIF _VarSetCmdParser.stCommand.ArrayType = DUT_Command_ArrayType.Flag THEN
				// will just let the flag take on the value of X
				SUPER^.Flags[_VarSetCmdParser.stCommand.ArrayIndex].Value := LREAL_TO_BOOL(_VarSetCmdParser.stCommand.Coordinates.X);
			END_IF
			// next, please
			SUPER^._SeqMain := _STEP_DONE;
			
		END_IF

END_CASE

METHOD PROTECTED M_Complete : BOOL
// once complete, reset to get back to idle
SUPER^._UnitMode.Reset();
END_METHOD

METHOD PROTECTED M_Execute : BOOL
// here we want to execute our commands/jobs/etc and set completed when done.
IF SUPER^._SeqMain =_STEP_IDLE THEN
	SUPER^.M_StateComplete();
END_IF
END_METHOD

METHOD PROTECTED M_SetPackML : BOOL
SUPER^._UnitMode(	sName := 'VarSet Processor', 
				eInitialState := PACK_ML.State.Idle,
				xActive := TRUE);
END_METHOD

METHOD PROTECTED M_Starting : BOOL
// here we want to clear things and get ready for the execute state
// I can consider this the "INIT" state
SUPER^._SeqMain := _STEP_COMMAND;
SUPER^.M_StateComplete();
END_METHOD

END_FUNCTION_BLOCK

// ---- FB/varset/ParseVarSetCmd.TcPOU
FUNCTION_BLOCK ParseVarSetCmd
VAR_INPUT
	Command: STRING(GVL.COMMAND_LEN);
END_VAR
VAR_OUTPUT
	stCommand: ST_VarSetCmd;
	Error: BOOL;
	ErrorDescription: STRING;
END_VAR
VAR
	_CmdParams: ARRAY [0..GVL.COMMAND_LEN] OF STRING;
END_VAR
VAR CONSTANT
	_ArrayTypeS: STRING(3):='STO';
	_ArrayTypeV: STRING(3):='VIS';
	_ArrayTypeF: STRING(3):='FLG';
END_VAR

// S|V|F index x y z a b c
// S 0000 +0000.00 +0000.00 +0000.00 +0000.00 +0000.00 +0000.00 
// V 0000 +0000.00 +0000.00 +0000.00 +0000.00 +0000.00 +0000.00 
// F 0000 1

Error:=FALSE;
ErrorDescription:='';

// split command string into commands
_CmdParams:=F_SplitCmd(Command:=Command);

//
IF _CmdParams[0] = _ArrayTypeS  THEN
	stCommand.ArrayType := DUT_Command_ArrayType.StoredPosition;
ELSIF _CmdParams[0] = _ArrayTypeV THEN
	stCommand.ArrayType := DUT_Command_ArrayType.VisionRegister;
ELSIF _CmdParams[0] = _ArrayTypeF THEN
	stCommand.ArrayType := DUT_Command_ArrayType.Flag;
ELSE
	Error:=TRUE;
	ErrorDescription:='Incorrect array type';
END_IF

//
stCommand.ArrayIndex := STRING_TO_INT(_CmdParams[1]);
IF ((stCommand.ArrayIndex < GVL.POS_ARR_BEG OR stCommand.ArrayIndex > GVL.POS_ARR_END) AND stCommand.ArrayType = DUT_Command_ArrayType.StoredPosition)
	OR ((stCommand.ArrayIndex < GVL.VIS_ARR_BEG OR stCommand.ArrayIndex > GVL.VIS_ARR_END) AND stCommand.ArrayType = DUT_Command_ArrayType.VisionRegister)
	OR ((stCommand.ArrayIndex < GVL.FLG_ARR_BEG OR stCommand.ArrayIndex > GVL.FLG_ARR_END) AND stCommand.ArrayType = DUT_Command_ArrayType.Flag) THEN
		Error:=TRUE;
		ErrorDescription:='Incorrect array type';
END_IF

//
stCommand.Coordinates.X := STRING_TO_LREAL(_CmdParams[2]);
stCommand.Coordinates.Y := STRING_TO_LREAL(_CmdParams[3]);
stCommand.Coordinates.Z := STRING_TO_LREAL(_CmdParams[4]);
stCommand.Coordinates.A := STRING_TO_LREAL(_CmdParams[5]);
stCommand.Coordinates.B := STRING_TO_LREAL(_CmdParams[6]);
stCommand.Coordinates.C := STRING_TO_LREAL(_CmdParams[7]);

END_FUNCTION_BLOCK

// ---- FB/logic/LogicCmdProcessor.TcPOU
FUNCTION_BLOCK LogicCmdProcessor EXTENDS Module
VAR_IN_OUT
	PrgProcessor: FB_ProgramProcessor;
	CmdProcessor: FB_CommandProcessor;
	CmdIO: ST_LogicCmdIO;
END_VAR
VAR_INPUT
	Command: STRING(GVL.COMMAND_LEN):='';
END_VAR
VAR_OUTPUT
END_VAR
VAR
	_UnitModeCurrentState: PACK_ML.State;
	_ParseLogicCmd: ParseLogicCmd;
	_ThenFunctionProcessed: BOOL;
END_VAR
VAR CONSTANT
	_STEP_DONE: 		INT := 1000;
	_STEP_IDLE: 		INT := 0000;
	_STEP_COMMAND: 		INT := 0010;
	_STEP_ERR: 			INT := 0020;
	_STEP_EVAL_IN:		INT := 0100;
	_STEP_EVAL_REG:		INT := 0110;
	_STEP_EVAL_CNT:		INT := 0120;
	_STEP_PROC_THEN:	INT := 0200;
	_STEP_PROC_ELSE:	INT := 0210;
	_STEP_PROC_OUT:		INT := 0300;
	_STEP_PROC_JMP:		INT := 0310;
	_STEP_PROC_CNT:		INT := 0320;
	_STEP_PROC_REG:		INT := 0330;
	_STEP_PROC_NOP:		INT := 0340;
	_STEP_PROC_CAL:		INT := 0350;
END_VAR

SUPER^();

// PackML state machine implementation
_UnitModeCurrentState := SUPER^._UnitMode.CurrentState;

//
CASE SUPER^._SeqMain OF
	
    _STEP_DONE:
		SUPER^._SeqMain := _STEP_IDLE;
        
    _STEP_IDLE:
		// wait here until commanded to start
        
    _STEP_COMMAND:
		_ParseLogicCmd(Command:=Command);
		
		CASE _ParseLogicCmd.stCommand.IF_Condition OF
			E_LogicIfCondition.PASS:
				SUPER^._SeqMain := _STEP_PROC_THEN;
			E_LogicIfCondition.INPUT:
				SUPER^._SeqMain := _STEP_EVAL_IN;
			E_LogicIfCondition.REGISTER:
				SUPER^._SeqMain := _STEP_EVAL_REG;
			E_LogicIfCondition.COUNTER:
				SUPER^._SeqMain := _STEP_EVAL_CNT;
		END_CASE
		
		//
		_ThenFunctionProcessed := FALSE;
		
	_STEP_EVAL_IN:
		CASE _ParseLogicCmd.stCommand.IF_Condition_Operator OF
			E_LogicIfConditionOperator.EQU:
				IF CmdIO.Input[_ParseLogicCmd.stCommand.IF_Condition_Idx] 
					= UDINT_TO_BOOL(_ParseLogicCmd.stCommand.IF_Condition_Operator_Value) THEN
						SUPER^._SeqMain := _STEP_PROC_THEN;
				ELSE
					SUPER^._SeqMain := _STEP_PROC_ELSE;
				END_IF
			E_LogicIfConditionOperator.GRE:
				IF CmdIO.Input[_ParseLogicCmd.stCommand.IF_Condition_Idx] 
					>= UDINT_TO_BOOL(_ParseLogicCmd.stCommand.IF_Condition_Operator_Value) THEN
						SUPER^._SeqMain := _STEP_PROC_THEN;
				ELSE
					SUPER^._SeqMain := _STEP_PROC_ELSE;
				END_IF
			E_LogicIfConditionOperator.GRT:
				IF CmdIO.Input[_ParseLogicCmd.stCommand.IF_Condition_Idx] 
					> UDINT_TO_BOOL(_ParseLogicCmd.stCommand.IF_Condition_Operator_Value) THEN
						SUPER^._SeqMain := _STEP_PROC_THEN;
				ELSE
					SUPER^._SeqMain := _STEP_PROC_ELSE;
				END_IF
			E_LogicIfConditionOperator.LEQ:
				IF CmdIO.Input[_ParseLogicCmd.stCommand.IF_Condition_Idx] 
					<= UDINT_TO_BOOL(_ParseLogicCmd.stCommand.IF_Condition_Operator_Value) THEN
						SUPER^._SeqMain := _STEP_PROC_THEN;
				ELSE
					SUPER^._SeqMain := _STEP_PROC_ELSE;
				END_IF
			E_LogicIfConditionOperator.LES:
				IF CmdIO.Input[_ParseLogicCmd.stCommand.IF_Condition_Idx] 
					< UDINT_TO_BOOL(_ParseLogicCmd.stCommand.IF_Condition_Operator_Value) THEN
						SUPER^._SeqMain := _STEP_PROC_THEN;
				ELSE
					SUPER^._SeqMain := _STEP_PROC_ELSE;
				END_IF
		END_CASE
		
	_STEP_EVAL_REG:
		CASE _ParseLogicCmd.stCommand.IF_Condition_Operator OF
			E_LogicIfConditionOperator.EQU:
				IF CmdIO.Register[_ParseLogicCmd.stCommand.IF_Condition_Idx] 
					= _ParseLogicCmd.stCommand.IF_Condition_Operator_Value THEN
						SUPER^._SeqMain := _STEP_PROC_THEN;
				ELSE
					SUPER^._SeqMain := _STEP_PROC_ELSE;
				END_IF
			E_LogicIfConditionOperator.GRE:
				IF CmdIO.Register[_ParseLogicCmd.stCommand.IF_Condition_Idx] 
					>= _ParseLogicCmd.stCommand.IF_Condition_Operator_Value THEN
						SUPER^._SeqMain := _STEP_PROC_THEN;
				ELSE
					SUPER^._SeqMain := _STEP_PROC_ELSE;
				END_IF
			E_LogicIfConditionOperator.GRT:
				IF CmdIO.Register[_ParseLogicCmd.stCommand.IF_Condition_Idx] 
					> _ParseLogicCmd.stCommand.IF_Condition_Operator_Value THEN
						SUPER^._SeqMain := _STEP_PROC_THEN;
				ELSE
					SUPER^._SeqMain := _STEP_PROC_ELSE;
				END_IF
			E_LogicIfConditionOperator.LEQ:
				IF CmdIO.Register[_ParseLogicCmd.stCommand.IF_Condition_Idx] 
					<= _ParseLogicCmd.stCommand.IF_Condition_Operator_Value THEN
						SUPER^._SeqMain := _STEP_PROC_THEN;
				ELSE
					SUPER^._SeqMain := _STEP_PROC_ELSE;
				END_IF
			E_LogicIfConditionOperator.LES:
				IF CmdIO.Register[_ParseLogicCmd.stCommand.IF_Condition_Idx] 
					< _ParseLogicCmd.stCommand.IF_Condition_Operator_Value THEN
						SUPER^._SeqMain := _STEP_PROC_THEN;
				ELSE
					SUPER^._SeqMain := _STEP_PROC_ELSE;
				END_IF
		END_CASE
		
	_STEP_EVAL_CNT:
		CASE _ParseLogicCmd.stCommand.IF_Condition_Operator OF
			E_LogicIfConditionOperator.EQU:
				IF CmdIO.Counter[_ParseLogicCmd.stCommand.IF_Condition_Idx] 
					= _ParseLogicCmd.stCommand.IF_Condition_Operator_Value THEN
						SUPER^._SeqMain := _STEP_PROC_THEN;
				ELSE
					SUPER^._SeqMain := _STEP_PROC_ELSE;
				END_IF
			E_LogicIfConditionOperator.GRE:
				IF CmdIO.Counter[_ParseLogicCmd.stCommand.IF_Condition_Idx] 
					>= _ParseLogicCmd.stCommand.IF_Condition_Operator_Value THEN
						SUPER^._SeqMain := _STEP_PROC_THEN;
				ELSE
					SUPER^._SeqMain := _STEP_PROC_ELSE;
				END_IF
			E_LogicIfConditionOperator.GRT:
				IF CmdIO.Counter[_ParseLogicCmd.stCommand.IF_Condition_Idx] 
					> _ParseLogicCmd.stCommand.IF_Condition_Operator_Value THEN
						SUPER^._SeqMain := _STEP_PROC_THEN;
				ELSE
					SUPER^._SeqMain := _STEP_PROC_ELSE;
				END_IF
			E_LogicIfConditionOperator.LEQ:
				IF CmdIO.Counter[_ParseLogicCmd.stCommand.IF_Condition_Idx] 
					<= _ParseLogicCmd.stCommand.IF_Condition_Operator_Value THEN
						SUPER^._SeqMain := _STEP_PROC_THEN;
				ELSE
					SUPER^._SeqMain := _STEP_PROC_ELSE;
				END_IF
			E_LogicIfConditionOperator.LES:
				IF CmdIO.Counter[_ParseLogicCmd.stCommand.IF_Condition_Idx] 
					< _ParseLogicCmd.stCommand.IF_Condition_Operator_Value THEN
						SUPER^._SeqMain := _STEP_PROC_THEN;
				ELSE
					SUPER^._SeqMain := _STEP_PROC_ELSE;
				END_IF
		END_CASE
		
	_STEP_PROC_THEN:
		//
		_ThenFunctionProcessed := TRUE;
		//
		CASE _ParseLogicCmd.stCommand.THEN_Function OF
			E_LogicFunction.OUTPUT:
				SUPER^._SeqMain := _STEP_PROC_OUT;
			E_LogicFunction.REGISTER:
				SUPER^._SeqMain := _STEP_PROC_REG;
			E_LogicFunction.CNTUP:
				SUPER^._SeqMain := _STEP_PROC_CNT;
			E_LogicFunction.CNTDN:
				SUPER^._SeqMain := _STEP_PROC_CNT;
			E_LogicFunction.CNTRST:
				SUPER^._SeqMain := _STEP_PROC_CNT;
			E_LogicFunction.JUMP:
				SUPER^._SeqMain := _STEP_PROC_JMP;
			E_LogicFunction.CALL:
				SUPER^._SeqMain := _STEP_PROC_CAL;
			E_LogicFunction.NOP:
				SUPER^._SeqMain := _STEP_PROC_NOP;
		END_CASE;
				
	_STEP_PROC_ELSE:
		CASE _ParseLogicCmd.stCommand.ELSE_Function OF
			E_LogicFunction.OUTPUT:
				SUPER^._SeqMain := _STEP_PROC_OUT;
			E_LogicFunction.REGISTER:
				SUPER^._SeqMain := _STEP_PROC_REG;
			E_LogicFunction.CNTUP:
				SUPER^._SeqMain := _STEP_PROC_CNT;
			E_LogicFunction.CNTDN:
				SUPER^._SeqMain := _STEP_PROC_CNT;
			E_LogicFunction.CNTRST:
				SUPER^._SeqMain := _STEP_PROC_CNT;
			E_LogicFunction.JUMP:
				SUPER^._SeqMain := _STEP_PROC_JMP;
			E_LogicFunction.CALL:
				SUPER^._SeqMain := _STEP_PROC_CAL;
			E_LogicFunction.NOP:
				SUPER^._SeqMain := _STEP_PROC_NOP;
		END_CASE;
		
	_STEP_PROC_OUT:
		IF _ThenFunctionProcessed THEN
			CmdIO.Output[_ParseLogicCmd.stCommand.THEN_Function_Idx] 
				:= UDINT_TO_BOOL(_ParseLogicCmd.stCommand.THEN_Function_Value);
		ELSE
			CmdIO.Output[_ParseLogicCmd.stCommand.ELSE_Function_Idx] 
				:= UDINT_TO_BOOL(_ParseLogicCmd.stCommand.ELSE_Function_Value);
		END_IF
		// next, please
		SUPER^._SeqMain := _STEP_DONE;
		
	_STEP_PROC_REG:
		IF _ThenFunctionProcessed THEN
			CmdIO.Register[_ParseLogicCmd.stCommand.THEN_Function_Idx] 
				:= _ParseLogicCmd.stCommand.THEN_Function_Value;
		ELSE
			CmdIO.Register[_ParseLogicCmd.stCommand.ELSE_Function_Idx] 
				:= _ParseLogicCmd.stCommand.ELSE_Function_Value;
		END_IF
		// next, please
		SUPER^._SeqMain := _STEP_DONE;
		
	_STEP_PROC_CNT:	
		IF _ThenFunctionProcessed THEN
			CASE _ParseLogicCmd.stCommand.THEN_Function OF
				E_LogicFunction.CNTUP:
					CmdIO.Counter[_ParseLogicCmd.stCommand.THEN_Function_Idx] 
						:= CmdIO.Counter[_ParseLogicCmd.stCommand.THEN_Function_Idx] + 1;
				E_LogicFunction.CNTDN:
					CmdIO.Counter[_ParseLogicCmd.stCommand.THEN_Function_Idx] 
						:= CmdIO.Counter[_ParseLogicCmd.stCommand.THEN_Function_Idx] - 1;
				E_LogicFunction.CNTRST:
					CmdIO.Counter[_ParseLogicCmd.stCommand.THEN_Function_Idx] 
						:= 0;
			END_CASE
		ELSE
			CASE _ParseLogicCmd.stCommand.ELSE_Function OF
				E_LogicFunction.CNTUP:
					CmdIO.Counter[_ParseLogicCmd.stCommand.ELSE_Function_Idx] 
						:= CmdIO.Counter[_ParseLogicCmd.stCommand.ELSE_Function_Idx] + 1;
				E_LogicFunction.CNTDN:
					CmdIO.Counter[_ParseLogicCmd.stCommand.ELSE_Function_Idx] 
						:= CmdIO.Counter[_ParseLogicCmd.stCommand.ELSE_Function_Idx] - 1;
				E_LogicFunction.CNTRST:
					CmdIO.Counter[_ParseLogicCmd.stCommand.ELSE_Function_Idx] 
						:= 0;
			END_CASE
		END_IF
		// next, please
		SUPER^._SeqMain := _STEP_DONE;
		
	_STEP_PROC_JMP:
		IF _ThenFunctionProcessed THEN
			CmdProcessor.M_SetNextCommand(CommandNumber:=INT_TO_UINT(_ParseLogicCmd.stCommand.THEN_Function_Idx));
		ELSE
			CmdProcessor.M_SetNextCommand(CommandNumber:=INT_TO_UINT(_ParseLogicCmd.stCommand.ELSE_Function_Idx));
		END_IF
		// next, please
		SUPER^._SeqMain := _STEP_DONE;
		
	_STEP_PROC_CAL:
		IF _ThenFunctionProcessed THEN
			PrgProcessor.M_CallProgram(	ProgramNumber:= INT_TO_UINT(_ParseLogicCmd.stCommand.THEN_Function_Idx), 
										ReturnProgram:= PrgProcessor.P_CurrentProgram, 
										ReturnCommand:= CmdProcessor.P_CurrentCommandIndex);
		ELSE
			PrgProcessor.M_CallProgram(	ProgramNumber:= INT_TO_UINT(_ParseLogicCmd.stCommand.ELSE_Function_Idx), 
										ReturnProgram:= PrgProcessor.P_CurrentProgram, 
										ReturnCommand:= CmdProcessor.P_CurrentCommandIndex);
		END_IF
		// next, please
		SUPER^._SeqMain := _STEP_DONE;
		
	_STEP_PROC_NOP:
		IF _ThenFunctionProcessed THEN
			//
		ELSE
			//
		END_IF
		// next, please
		SUPER^._SeqMain := _STEP_DONE;

END_CASE

METHOD PROTECTED M_Complete : BOOL
// once complete, reset to get back to idle
SUPER^._UnitMode.Reset();
END_METHOD

METHOD PROTECTED M_Execute : BOOL
// here we want to execute our commands/jobs/etc and set completed when done.
IF SUPER^._SeqMain =_STEP_IDLE THEN
	SUPER^.M_StateComplete();
END_IF
END_METHOD

METHOD PROTECTED M_SetPackML : BOOL
SUPER^._UnitMode(	sName := 'Logic Processor',
				eInitialState := PACK_ML.State.Idle,
				xActive := TRUE);
END_METHOD

METHOD PROTECTED M_Starting : BOOL
// here we want to clear things and get ready for the execute state
// I can consider this the "INIT" state
SUPER^._SeqMain := _STEP_COMMAND;
SUPER^.M_StateComplete();
END_METHOD

END_FUNCTION_BLOCK

// ---- FB/logic/ParseLogicCmd.TcPOU
FUNCTION_BLOCK ParseLogicCmd
VAR_INPUT
	Command: STRING(GVL.COMMAND_LEN);
END_VAR
VAR_OUTPUT
	stCommand: ST_LogicCmd;
	Error: BOOL;
	ErrorDescription: STRING;
END_VAR
VAR
	_CmdParams: ARRAY [0..GVL.COMMAND_LEN] OF STRING;
	_i, _j, _k: INT;
END_VAR

// IF PASS|INPUT|REGISTER|COUNTER <index> >|<|=|>=|<= <value>
// THEN OUTPUT|JUMP|CALL|CNTUP|CNTDN|CNTRST|REGISTER|NOP <index> <value>
// ELSE OUTPUT|JUMP|CALL|CNTUP|CNTDN|CNTRST|REGISTER|NOP <index> <value>
//
// IF_Condition
// IF_Condition_Idx
// IF_Condition_Operator
// IF_Condition_Operator_Compare
// THEN_Function
// THEN_Function_Value
// THEN_Function_Idx
// ELSE_Function
// ELSE_Function_Idx
// ELSE_Function_Value

Error:=FALSE;
ErrorDescription:='';

// split command string into commands
_CmdParams:=F_SplitCmd(Command:=Command);

//
_i := 0;

// disregard the 'IF'
_i := _i + 1;

//
IF _CmdParams[_i] = TO_STRING(E_LogicIfCondition.PASS) THEN
	stCommand.IF_Condition := E_LogicIfCondition.PASS;
ELSIF  _CmdParams[_i] = TO_STRING(E_LogicIfCondition.INPUT) THEN
	stCommand.IF_Condition := E_LogicIfCondition.INPUT;
ELSIF  _CmdParams[_i] = TO_STRING(E_LogicIfCondition.REGISTER) THEN
	stCommand.IF_Condition := E_LogicIfCondition.REGISTER;
ELSIF  _CmdParams[_i] = TO_STRING(E_LogicIfCondition.COUNTER) THEN
	stCommand.IF_Condition := E_LogicIfCondition.COUNTER;
END_IF
_i := _i + 1;

//
IF stCommand.IF_Condition <> E_LogicIfCondition.PASS THEN
	
	//
	stCommand.IF_Condition_Idx := STRING_TO_INT(_CmdParams[_i]);
	_i := _i + 1;
	
	//
	IF _CmdParams[_i] = TO_STRING(E_LogicIfConditionOperator.GRT) THEN
		stCommand.IF_Condition_Operator := E_LogicIfConditionOperator.GRT;
	ELSIF _CmdParams[_i] = TO_STRING(E_LogicIfConditionOperator.LES) THEN
		stCommand.IF_Condition_Operator := E_LogicIfConditionOperator.LES;                   
	ELSIF _CmdParams[_i] = TO_STRING(E_LogicIfConditionOperator.EQU) THEN
		stCommand.IF_Condition_Operator := E_LogicIfConditionOperator.EQU;
	ELSIF _CmdParams[_i] = TO_STRING(E_LogicIfConditionOperator.GRE) THEN
		stCommand.IF_Condition_Operator := E_LogicIfConditionOperator.GRE;
	ELSIF _CmdParams[_i] = TO_STRING(E_LogicIfConditionOperator.LEQ) THEN
		stCommand.IF_Condition_Operator := E_LogicIfConditionOperator.LEQ;
	END_IF
	_i := _i + 1;
	
	//
	stCommand.IF_Condition_Operator_Value := STRING_TO_UDINT(_CmdParams[_i]);
	_i := _i + 1;
	
END_IF

// disregard the 'THEN'
_i := _i + 1;

//
IF _CmdParams[_i] = TO_STRING(E_LogicFunction.OUTPUT) THEN
	stCommand.THEN_Function := E_LogicFunction.OUTPUT;
ELSIF _CmdParams[_i] = TO_STRING(E_LogicFunction.JUMP) THEN
	stCommand.THEN_Function := E_LogicFunction.JUMP;
ELSIF _CmdParams[_i] = TO_STRING(E_LogicFunction.CALL) THEN
	stCommand.THEN_Function := E_LogicFunction.CALL;           
ELSIF _CmdParams[_i] = TO_STRING(E_LogicFunction.CNTUP) THEN
	stCommand.THEN_Function := E_LogicFunction.CNTUP;
ELSIF _CmdParams[_i] = TO_STRING(E_LogicFunction.CNTDN) THEN
	stCommand.THEN_Function := E_LogicFunction.CNTDN;
ELSIF _CmdParams[_i] = TO_STRING(E_LogicFunction.CNTRST) THEN
	stCommand.THEN_Function := E_LogicFunction.CNTRST;
ELSIF _CmdParams[_i] = TO_STRING(E_LogicFunction.REGISTER) THEN
	stCommand.THEN_Function := E_LogicFunction.REGISTER;
ELSIF _CmdParams[_i] = TO_STRING(E_LogicFunction.NOP) THEN
	stCommand.THEN_Function := E_LogicFunction.NOP;
END_IF
_i := _i + 1;

//
IF stCommand.THEN_Function <> E_LogicFunction.NOP THEN
	stCommand.THEN_Function_Idx := STRING_TO_INT(_CmdParams[_i]);
	_i := _i + 1;
	IF stCommand.THEN_Function = E_LogicFunction.OUTPUT 
		OR stCommand.THEN_Function = E_LogicFunction.REGISTER THEN
			stCommand.THEN_Function_Value := STRING_TO_UDINT(_CmdParams[_i]);
			_i := _i + 1;
	END_IF
END_IF

// disregard the 'ELSE'
_i := _i + 1;

//
IF _CmdParams[_i] = TO_STRING(E_LogicFunction.OUTPUT) THEN
	stCommand.ELSE_Function := E_LogicFunction.OUTPUT;
ELSIF _CmdParams[_i] = TO_STRING(E_LogicFunction.JUMP) THEN
	stCommand.ELSE_Function := E_LogicFunction.JUMP;
ELSIF _CmdParams[_i] = TO_STRING(E_LogicFunction.CALL) THEN
	stCommand.ELSE_Function := E_LogicFunction.CALL;
ELSIF _CmdParams[_i] = TO_STRING(E_LogicFunction.CNTUP) THEN
	stCommand.ELSE_Function := E_LogicFunction.CNTUP;
ELSIF _CmdParams[_i] = TO_STRING(E_LogicFunction.CNTDN) THEN
	stCommand.ELSE_Function := E_LogicFunction.CNTDN;
ELSIF _CmdParams[_i] = TO_STRING(E_LogicFunction.CNTRST) THEN
	stCommand.ELSE_Function := E_LogicFunction.CNTRST;
ELSIF _CmdParams[_i] = TO_STRING(E_LogicFunction.REGISTER) THEN
	stCommand.ELSE_Function := E_LogicFunction.REGISTER;
ELSIF _CmdParams[_i] = TO_STRING(E_LogicFunction.NOP) THEN
	stCommand.ELSE_Function := E_LogicFunction.NOP;
END_IF
_i := _i + 1;

//
IF stCommand.ELSE_Function <> E_LogicFunction.NOP THEN
	stCommand.ELSE_Function_Idx := STRING_TO_INT(_CmdParams[_i]);
	_i := _i + 1;
	IF stCommand.ELSE_Function = E_LogicFunction.OUTPUT 
		OR stCommand.ELSE_Function = E_LogicFunction.REGISTER THEN
			stCommand.ELSE_Function_Value := STRING_TO_UDINT(_CmdParams[_i]);
			_i := _i + 1;
	END_IF
END_IF

END_FUNCTION_BLOCK

// ---- FB/digital/FB_DigitalOutput.TcPOU
FUNCTION_BLOCK FB_DigitalOutput
VAR_INPUT
END_VAR
VAR_OUTPUT
END_VAR
VAR	
	// https://infosys.beckhoff.com/content/1033/tc3_plc_intro/11948825611.html?id=1756449079294237528
	Output AT %Q* : BOOL;
	_Output: BOOL;
	_FirstScan: BOOL;
END_VAR

IF _FirstScan THEN
	//
END_IF

// do some things?
Output :=_Output;

// do not put anything below this
_FirstScan := FALSE;

METHOD PUBLIC Off : BOOL
VAR_INPUT
END_VAR
_Output := FALSE;
END_METHOD

METHOD PUBLIC On : BOOL
VAR_INPUT
END_VAR
_Output := TRUE;
END_METHOD

{attribute 'monitoring' := 'variable'}
PROPERTY PUBLIC P_StateOff : BOOL
GET
P_StateOff := NOT _Output;
END_GET
END_PROPERTY

{attribute 'monitoring' := 'variable'}
PROPERTY PUBLIC P_StateOn : BOOL
GET
P_StateOn := _Output;
END_GET
END_PROPERTY

METHOD PUBLIC Toggle : BOOL
VAR_INPUT
END_VAR
_Output := NOT _Output;
END_METHOD

END_FUNCTION_BLOCK

// ---- FB/controller/FB_Controller.TcPOU
FUNCTION_BLOCK FB_Controller EXTENDS PythonServerHandler
VAR_INPUT
END_VAR
VAR_OUTPUT
END_VAR
VAR
	Controller: ST_Controller;
	ControllerStates: ARRAY [0..254] OF BYTE;
	ControllerStatesTemp: ARRAY [0..254] OF BYTE;
	ReadStringTemp: STRING(255);
	RecordLast: DINT;
	ReconnectTimer: TON:=(PT:=T#5S);
	
	_SetColor: BOOL;
	_Red: INT:=0;
	_Green: INT:=255;
	_Blue: INT:=0;
	
	_SetMicrophoneState: BOOL;
	_MicrophoneState: BOOL;
	
	_SetPlayerID: BOOL;
	_PlayerID: E_ControllerPlayerID;
	
	_SetBrightness: BOOL;
	_Brightness: E_ControllerBrightness;
	
	_SetMotorIntensity: BOOL;
	_Motor: E_ControllerMotor;
	_MotorIntensity: USINT; // 0-255
	_MotorIntensityDuration: REAL; // ms
	
	_SetTriggerMode: BOOL;
	_TriggerModeTrigger: E_ControllerTrigger;
	_TriggerModeMode: E_ControllerTriggerMode;
	
	_SetTriggerForce: BOOL;
	_TriggerForceTrigger: E_ControllerTrigger;
	_TriggerForceParameter: E_ControllerTriggerForceParameter;
	_TriggerForceIntensity: USINT;
	
	_i, _j, _k: INT;
	FirstScan: BOOL:=TRUE;
END_VAR
VAR CONSTANT
	States: STRING:='states: ';
END_VAR

SUPER^();

// copy over controller states when a new message is received
IF SUPER^.P_RecordNumber <> RecordLast THEN
	RecordLast := SUPER^.P_RecordNumber;
	IF FIND(SUPER^.P_RawReadString, States) > 0 THEN // TODO this is getting messy. need to overhaul how this works
		ControllerStatesTemp := SUPER^.P_RawReadByteArray;
		FOR _i:=0 TO UINT_TO_INT(SIZEOF(ControllerStates)) - LEN(States) BY 1 DO
			ControllerStates[_i] := ControllerStatesTemp[_i + LEN(States)];
		END_FOR
		
	END_IF
END_IF

//
_M_EvaluateControllerStates(States:=ControllerStates);
_M_SetColor();
_M_SetMicrophoneState();
_M_SetPlayerID();
_M_SetBrightness();
_M_SetMotorIntensity();
_M_SetTriggerMode();
_M_SetTriggerForce();

// try to reconnect to the server when data stops?
// leave this commented out until we have a better condition
// the edge case is when the controller is connected via bluetooth 
// but for some reason the server is not connected to it.
// maybe work this issue out on the server side.
(*ReconnectTimer(IN:= RecordLast=SUPER^.P_RecordNumber);
IF ReconnectTimer.Q THEN
	ReconnectTimer(IN:=FALSE);
	SUPER^.M_Reconnect();
END_IF*)

FirstScan:=FALSE;

METHOD PRIVATE _M_EvaluateControllerStates : BOOL
VAR_INPUT
	States: ARRAY[0..254] OF BYTE;
END_VAR
VAR_STAT
	_i: UINT;
	_j: UINT;
	_k: UINT;
	_FirstScan: BOOL := TRUE;
	_HeartbeatTimer: TON := (PT := TIME#2s0ms);
	_Heartbeat: USINT := 0;
	_HeartbeatLast: USINT := 0;
END_VAR
IF _FirstScan THEN
	//
END_IF

//
_Heartbeat := States[0] OR States[7]; // States[0] appears to be bluetooth and States[7] appears to be wired
IF _Heartbeat <> _HeartbeatLast THEN
	_HeartbeatLast := _Heartbeat;
	_HeartbeatTimer(IN:=FALSE);
ELSE
	_HeartbeatTimer(IN:=TRUE);
END_IF
Controller.Connected S= NOT _HeartbeatTimer.IN;
Controller.Connected R= _HeartbeatTimer.Q;

// clear all the data if the controller disconnects
IF NOT Controller.Connected THEN
	//MemUtils.MemSet(pbyBuffer:=ADR(States), byValue:=0, dwSize:=SIZEOF(States)); 
	FOR _i:=1 TO 254 BY 1 DO // start at 1 so we dont overwrite the heartbeat
		States[_i] := 0;
	END_FOR
END_IF

Controller.Joysticks.Left.X					:= States[1];
Controller.Joysticks.Left.Y					:= States[2];
Controller.Joysticks.Right.X				:= States[3];
Controller.Joysticks.Right.Y				:= States[4];
Controller.Triggers.Left.Two				:= States[5];
Controller.Triggers.Right.Two				:= States[6];

//UNUSED									:= States[7];

Controller.Buttons.Triangle 				:= States[8].7;
Controller.Buttons.Circle 					:= States[8].6;
Controller.Buttons.Cross 					:= States[8].5;
Controller.Buttons.Square 					:= States[8].4;
Controller.Dpad								:= F_DpadState(States[8] AND 16#0F);

Controller.Joysticks.Right.ThreeButton 		:= States[9].7;
Controller.Joysticks.Left.ThreeButton 		:= States[9].6;
Controller.Buttons.Options 					:= States[9].5;
Controller.Buttons.Share 					:= States[9].4;
Controller.Triggers.Right.TwoButton 		:= States[9].3;
Controller.Triggers.Left.TwoButton 			:= States[9].2;
Controller.Triggers.Right.One 				:= States[9].1;
Controller.Triggers.Left.One 				:= States[9].0;

Controller.Buttons.PS						:= States[10].0;
Controller.Buttons.Touch					:= States[10].1;
Controller.Buttons.Mic						:= States[10].2;

//UNUSED									:= States[11];
//UNUSED									:= States[12];
//UNUSED									:= States[13];
//UNUSED									:= States[14];
//UNUSED									:= States[15];

Controller.Accelerometer.X					:= SHL(States[16], 8) OR States[17];
Controller.Accelerometer.Y					:= SHL(States[18], 8) OR States[19];
Controller.Accelerometer.Z					:= SHL(States[20], 8) OR States[21];

Controller.Gyroscope.Pitch					:= SHL(States[22], 8) OR States[23];
Controller.Gyroscope.Yaw					:= SHL(States[24], 8) OR States[25];
Controller.Gyroscope.Roll					:= SHL(States[26], 8) OR States[27];

//UNUSED									:= States[28];
//UNUSED									:= States[29];
//UNUSED									:= States[30];
//UNUSED									:= States[31];
//UNUSED									:= States[32];

Controller.Trackpads.One.ID					:= States[33] AND 16#7F;
Controller.Trackpads.One.Active				:= (States[33] AND 16#80) = 0;
Controller.Trackpads.One.X					:= SHL((States[35] AND 16#0F), 8) OR States[34];
Controller.Trackpads.One.Y					:= SHL(States[36], 4) OR SHR((States[35] AND 16#F0), 4);
Controller.Trackpads.Two.ID					:= States[37] AND 16#7F;
Controller.Trackpads.Two.Active				:= (States[37] AND 16#80) = 0;
Controller.Trackpads.Two.X					:= SHL((States[39] AND 16#0F), 8) OR States[38];
Controller.Trackpads.Two.Y					:= SHL(States[40], 4) OR SHR((States[39] AND 16#F0), 4);

//UNUSED									:= States[41];
//UNUSED									:= States[42];
//UNUSED									:= States[43];
//UNUSED									:= States[44];
//UNUSED									:= States[45];
//UNUSED									:= States[46];
//UNUSED									:= States[47];
//UNUSED									:= States[48];
//UNUSED									:= States[49];
//UNUSED									:= States[50];
//UNUSED									:= States[51];
//UNUSED									:= States[52];

// from kit-nya
Controller.Battery.State					:= SHR(States[53] AND 16#F0, 4);
Controller.Battery.Level					:= MIN((States[53] AND 16#0F) * 10 + 5, 100); // TODO this will show a value of 5 when controller is disconnected.

// dont put anything below this
_FirstScan := FALSE;
END_METHOD

METHOD PRIVATE _M_SetBrightness : BOOL
IF NOT SUPER^._Busy AND _SetBrightness THEN
	_SetBrightness := FALSE;
	
	_Command := CONCAT('cmd: setBrightness:', INT_TO_STRING(_Brightness));
	
	SUPER^._M_Execute(Command:=_Command, Timeout:=5);
	SUPER^(); // call super here so other methods see it busy.
END_IF
END_METHOD

METHOD PRIVATE _M_SetColor : BOOL
VAR
	_Command: STRING(255);
END_VAR
IF NOT SUPER^._Busy AND_THEN _SetColor THEN
	_SetColor := FALSE;
	
	_Command := CONCAT('cmd: setColorI:', INT_TO_STRING(_Red));
	_Command := CONCAT(_Command, ',');
	_Command := CONCAT(_Command, INT_TO_STRING(_Green));
	_Command := CONCAT(_Command, ',');
	_Command := CONCAT(_Command, INT_TO_STRING(_Blue));
	
	SUPER^._M_Execute(Command:=_Command, Timeout:=5);
	SUPER^(); // call super here so other methods see it busy.
END_IF
END_METHOD

METHOD PRIVATE _M_SetMicrophoneState : BOOL
VAR
	_Command: STRING(255);
END_VAR
IF NOT SUPER^._Busy AND _SetMicrophoneState THEN
	_SetMicrophoneState := FALSE;
	
	_Command := CONCAT('cmd: setMicrophoneState:', BOOL_TO_STRING(_MicrophoneState));
	
	SUPER^._M_Execute(Command:=_Command, Timeout:=5);
	SUPER^(); // call super here so other methods see it busy.
END_IF;
END_METHOD

METHOD PRIVATE _M_SetMotorIntensity : BOOL
VAR
	_Command: STRING(255);
END_VAR
IF NOT SUPER^._Busy AND _SetMotorIntensity THEN
	_SetMotorIntensity := FALSE;
	
	IF _Motor = E_ControllerMotor.Left THEN
		_Command := 'cmd: setLeftMotor:';
	ELSE
		_Command := 'cmd: setRightMotor:';
	END_IF
	_Command := CONCAT(_Command, USINT_TO_STRING(_MotorIntensity));
	_Command := CONCAT(_Command, ',');
	_Command := CONCAT(_Command, REAL_TO_STRING(_MotorIntensityDuration));
	
	SUPER^._M_Execute(Command:=_Command, Timeout:=5);
	SUPER^(); // call super here so other methods see it busy.
END_IF
END_METHOD

METHOD PRIVATE _M_SetPlayerID : BOOL
VAR
	_Command: STRING(255);
END_VAR
IF NOT SUPER^._Busy AND _SetPlayerID THEN
	_SetPlayerID := FALSE;
	
	_Command := CONCAT('cmd: setPlayerID:', INT_TO_STRING(_PlayerID));
	
	SUPER^._M_Execute(Command:=_Command, Timeout:=5);
	SUPER^(); // call super here so other methods see it busy.
END_IF
END_METHOD

METHOD PRIVATE _M_SetTriggerForce : BOOL
VAR
	_Command: STRING(255);
END_VAR

IF NOT SUPER^._Busy AND _SetTriggerForce THEN
	_SetTriggerForce := FALSE;
	
	IF _TriggerForceTrigger = E_ControllerTrigger.Left THEN
		_Command := 'cmd: setLeftTriggerForce:';
	ELSE
		_Command := 'cmd: setRightTriggerForce:';
	END_IF
	_Command := CONCAT(_Command, INT_TO_STRING(_TriggerForceParameter));
	_Command := CONCAT(_Command, ',');
	_Command := CONCAT(_Command, USINT_TO_STRING(_TriggerForceIntensity));
	
	SUPER^._M_Execute(Command:=_Command, Timeout:=5);
	SUPER^(); // call super here so other methods see it busy.
END_IF
END_METHOD

METHOD PRIVATE _M_SetTriggerMode : BOOL
VAR
	_Command: STRING(255);
END_VAR

IF NOT SUPER^._Busy AND _SetTriggerMode THEN
	_SetTriggerMode := FALSE;
	
	IF _TriggerModeTrigger = E_ControllerTrigger.Left THEN
		_Command := 'cmd: setLeftTriggerMode:';
	ELSE
		_Command := 'cmd: setRightTriggerMode:';
	END_IF
	_Command := CONCAT(_Command, INT_TO_STRING(_TriggerModeMode));
	
	SUPER^._M_Execute(Command:=_Command, Timeout:=5);
	SUPER^(); // call super here so other methods see it busy.
END_IF
END_METHOD

METHOD M_SetBrightness : BOOL
VAR_INPUT
	Brightness: E_ControllerBrightness;
END_VAR
M_SetBrightness := TRUE;
_Brightness := Brightness;
_SetBrightness := TRUE;
END_METHOD

METHOD M_SetColor : BOOL
VAR_INPUT
	Red: INT := 0;
	Green: INT := 255;
	Blue: INT := 0;
END_VAR
IF Red>=0 AND_THEN Red<=255
	AND_THEN Green>=0 AND_THEN Green<=255
	AND_THEN Blue>=0 AND_THEN Blue<=255THEN
		M_SetColor := TRUE;
		_SetColor:=TRUE;
		_Red:=Red;
		_Green:=Green;
		_Blue:=Blue;
ELSE
	M_SetColor := FALSE;
END_IF
END_METHOD

METHOD M_SetMicrophoneState : BOOL
VAR_INPUT
	State: BOOL;
END_VAR
M_SetMicrophoneState := TRUE;
_MicrophoneState := State;
_SetMicrophoneState := TRUE;
END_METHOD

METHOD M_SetMotorIntensity : BOOL
VAR_INPUT
	Motor: E_ControllerMotor;
	/// 0-255
	Intensity: USINT;
	/// s
	Duration: REAL;
END_VAR
IF Intensity >=0 AND_THEN Intensity <= 255 AND_THEN Duration <= 5000 THEN
	M_SetMotorIntensity := TRUE;
	_SetMotorIntensity := TRUE;
	_Motor := Motor;
	_MotorIntensity := Intensity;
	_MotorIntensityDuration := Duration;
ELSE
	M_SetMotorIntensity := FALSE;
END_IF
END_METHOD

METHOD M_SetPlayerID : BOOL
VAR_INPUT
	PlayerID: E_ControllerPlayerID;
END_VAR
M_SetPlayerID := TRUE;
_PlayerID := PlayerID;
_SetPlayerID := TRUE;
END_METHOD

METHOD M_SetTriggerForce : BOOL
VAR_INPUT
	Trigger: E_ControllerTrigger;
	Parameter: E_ControllerTriggerForceParameter;
	/// 0-255
	Intensity: USINT;
END_VAR
IF Intensity >= 0 AND Intensity <= 255 THEN
	M_SetTriggerForce := TRUE;
	_SetTriggerForce:=TRUE;
	_TriggerForceTrigger := Trigger;
	_TriggerForceParameter := Parameter;
	_TriggerForceIntensity := Intensity;
ELSE
	M_SetTriggerForce := FALSE;
END_IF
END_METHOD

METHOD M_SetTriggerMode : BOOL
VAR_INPUT
	Trigger: E_ControllerTrigger;
	Mode: E_ControllerTriggerMode;
END_VAR
M_SetTriggerMode := TRUE;
_SetTriggerMode := TRUE;
_TriggerModeTrigger := Trigger;
_TriggerModeMode := Mode;
END_METHOD

{attribute 'monitoring' := 'variable'}
PROPERTY P_State : REFERENCE TO ST_Controller
GET
P_State REF= Controller;
END_GET
END_PROPERTY

END_FUNCTION_BLOCK

// ---- FB/tcp/PythonServerHandler.TcPOU
FUNCTION_BLOCK PythonServerHandler
VAR_INPUT
	sIpAddress: STRING(19):='127.0.0.1';
	uPort: UINT:=50011;
END_VAR
VAR_OUTPUT
END_VAR
VAR
	_Done: BOOL;
	_Busy: BOOL;
	_Error: BOOL;
	_ErrorDescription: STRING;
	_Response: STRING(255);
	_WorkerUid: STRING;
	_Execute: BOOL;
	_Reset: BOOL:=FALSE;
	_ResetRtrig: R_TRIG;
	_Step: INT;
	_Command: STRING(255);
	_ReadRecordLast: DINT;
	_TcpClient: TcpClient;
	_TimeoutTimer: TON:=(PT:=T#120S);
END_VAR

_TimeoutTimer(IN:=_Step > 0);
IF _TimeoutTimer.Q THEN
	_Step := 0;
	_Error := TRUE;
	_ErrorDescription := 'timed out waiting for response.';
END_IF

_ResetRtrig(CLK:=_Reset);
IF _ResetRtrig.Q THEN
	_Reset := FALSE;
	_Step := 0;
END_IF

_Done := _Step = 0;
_Busy := NOT _Done;

CASE _Step OF
	0: // IDLE
		IF _Execute THEN
			_Execute := FALSE;
			IF _TcpClient._M_Write(Data:=_Command) THEN
				_ReadRecordLast := _TcpClient.dRecordRead;
				_Step := _Step + 1;
			ELSE
				_Step := 0;
			END_IF
		END_IF
	
	1: // WAIT
		IF _TcpClient.dRecordRead <> _ReadRecordLast THEN
			_ReadRecordLast := _TcpClient.dRecordRead;
			IF find(_TcpClient.strRead, 'res: ') = 1 THEN
				MemSet(
					destAddr:=ADR(_Response),
					fillByte:=0,
					n:=SIZEOF(_Response));
				_Response := _TcpClient.strRead;
				_Step := 0;
				
			ELSIF find(_TcpClient.strRead, 'worker uid: ') = 1 THEN
				MemSet(
					destAddr:=ADR(_WorkerUid),
					fillByte:=0,
					n:=SIZEOF(_WorkerUid));
				_WorkerUid := DELETE(STR:=_TcpClient.strRead, LEN:=12, POS:=1);
				
			ELSIF find(_TcpClient.strRead, 'command uid: ') = 1 THEN
				MemSet(
					destAddr:=ADR(_WorkerUid),
					fillByte:=0,
					n:=SIZEOF(_WorkerUid));
				_WorkerUid := DELETE(STR:=_TcpClient.strRead, LEN:=12, POS:=1);
				
			END_IF
		END_IF
		
END_CASE

_TcpClient(
	bEnable:= TRUE, 
	strIpAddress:= sIpAddress, 
	uPort:= uPort,
	bBusyWrite=> , 
	bDoneWrite=> , 
	bBusyRead=> , 
	dRecordRead=> , 
	strRead=> );

METHOD PROTECTED _M_Execute : BOOL
VAR_INPUT
	Command: STRING(255) := '';
	Timeout: UDINT := 60;
END_VAR
_Execute := TRUE;
_Command:=Command;
_TimeoutTimer.PT := UDINT_TO_TIME(Timeout * 1000);
END_METHOD

METHOD M_Cancel : BOOL
IF _WorkerUid <> '' THEN
	M_Cancel := TRUE;
	_Command := 'kill: ';
	_Command := CONCAT(_Command, _WorkerUid);
	_WorkerUid := ''; // lets make sure to forget this uid in case its used again for something else
	_Step := 0;
	_Execute := TRUE;
	
ELSE
	M_Cancel := FALSE;
	
END_IF
END_METHOD

METHOD M_Reconnect : BOOL
_TcpClient._M_Reconnect();
END_METHOD

METHOD M_Reset : BOOL
_Reset := TRUE;
_Error := FALSE;
_ErrorDescription := '';
END_METHOD

{attribute 'monitoring' := 'variable'}
PROPERTY P_Busy : BOOL
GET
P_Busy := _Busy;
END_GET
END_PROPERTY

{attribute 'monitoring' := 'variable'}
PROPERTY P_Connected : REFERENCE TO BOOL
GET
P_Connected REF= _TcpClient.bConnected;
END_GET
END_PROPERTY

{attribute 'monitoring' := 'variable'}
PROPERTY P_Done : BOOL
GET
P_Done := _Done;
END_GET
END_PROPERTY

{attribute 'monitoring' := 'variable'}
PROPERTY P_Error : BOOL
GET
P_Error := _Error;
END_GET
END_PROPERTY

{attribute 'monitoring' := 'variable'}
PROPERTY P_ErrorDescription : STRING
GET
P_ErrorDescription := _ErrorDescription;
END_GET
END_PROPERTY

{attribute 'monitoring' := 'variable'}
PROPERTY P_RawReadByteArray : ARRAY[0..254] OF BYTE
GET
P_RawReadByteArray := _TcpClient.byteArrayRead;
END_GET
END_PROPERTY

{attribute 'monitoring' := 'variable'}
PROPERTY P_RawReadString : REFERENCE TO STRING(255)
GET
P_RawReadString REF= _TcpClient.strRead;
END_GET
END_PROPERTY

{attribute 'monitoring' := 'variable'}
PROPERTY P_RecordNumber : DINT
GET
P_RecordNumber := _TcpClient.dRecordRead;
END_GET
END_PROPERTY

{attribute 'monitoring' := 'variable'}
PROPERTY P_Response : STRING(255)
GET
P_Response := _Response;
END_GET
END_PROPERTY

END_FUNCTION_BLOCK

// ---- FB/tcp/TcpClient.TcPOU
FUNCTION_BLOCK TcpClient
VAR_INPUT
	bEnable: BOOL;
	strIpAddress: STRING(19):='127.0.0.1';
	uPort: UINT:=50011;
END_VAR
VAR
	_Write: BOOL:=FALSE;
	_DataToWrite: STRING(255):='';
END_VAR
VAR_OUTPUT
	bBusyWrite: BOOL;
	bDoneWrite: BOOL;
	bBusyRead: BOOL;
	dRecordRead: DINT;
	strRead: STRING(255);
	byteArrayRead: ARRAY[0..254] OF BYTE;
	bConnected: BOOL;
END_VAR

VAR
    _ipAddress       : NBS.IPv4Address;
    _fbTcpClient     : NBS.TCP_Client;
    _fbTcpRead       : NBS.TCP_Read;
    _fbTcpWrite      : NBS.TCP_Write;	
	
	_ConnectDelayTimer: TON;
	
	_WriteData: StringByteArray;
	_ReadData: StringByteArray;
	
	_WriteRTRIG: R_TRIG;
	_ConnectStep, _ReadStep: INT;
	_Read: BOOL;
END_VAR

VAR CONSTANT
	ConnectStep_IDLE: 	INT:=00;
	ConnectStep_DELAY: 	INT:=10;
	ConnectStep_SETUP: 	INT:=20;
	ConnectStep_ENABLE: INT:=30;
	ConnectStep_WAIT: 	INT:=40;
	ConnectStep_CONN: 	INT:=50;
END_VAR

VAR CONSTANT
	WriteStep_IDLE: 	INT:=00;
	WriteStep_DATA: 	INT:=10;
	WriteStep_WRITE: 	INT:=20;
	WriteStep_WAIT: 	INT:=30;
END_VAR

VAR CONSTANT
	ReadStep_RESET: 	INT:=00;
	ReadStep_IDLE: 		INT:=10;
	ReadStep_ENABLE: 	INT:=20;
	ReadStep_MONITOR: 	INT:=30;
END_VAR

{region "connect"}
	
	bConnected := (_ConnectStep = ConnectStep_CONN);
	_ConnectDelayTimer(IN:=_ConnectStep = ConnectStep_DELAY, PT:=T#1S);
	CASE _ConnectStep OF
		
		ConnectStep_IDLE: // IDLE
			IF bEnable THEN
				_fbTcpClient.xEnable := FALSE;
				_ConnectStep := ConnectStep_DELAY;
			END_IF
			
		ConnectStep_DELAY: // DELAY
			IF _ConnectDelayTimer.Q THEN
				_ConnectStep := ConnectStep_SETUP;
			END_IF
			
		ConnectStep_SETUP: // SETUP
			_ipAddress.SetInitialValue(ipAddress := strIpAddress);
			_ConnectStep := ConnectStep_ENABLE;
			
		ConnectStep_ENABLE: // ENABLE
			_fbTcpClient.xEnable := TRUE;
			_ConnectStep := ConnectStep_WAIT;
			
		ConnectStep_WAIT: // WAIT
			IF _fbTcpClient.xActive THEN
				_ConnectStep := ConnectStep_CONN;
			ELSIF _fbTcpClient.xError THEN
				_ConnectStep := ConnectStep_IDLE;
			END_IF
		
		ConnectStep_CONN: // CONNECTED
			IF _fbTcpClient.xError OR NOT _fbTcpClient.xActive OR NOT bEnable THEN
				_ConnectStep := ConnectStep_IDLE;
			END_IF
			
	END_CASE
	
	_fbTcpClient(
		xEnable := , 
		itfIPAddress := _ipAddress, 
		uiPort := uPort, 
		udiTimeOut := 1000000); // us
			 
{endregion}


{region "write"}
	_WriteRTRIG(CLK:=_Write);
	IF _WriteRTRIG.Q THEN
		_Write := FALSE;
		IF bConnected AND _DataToWrite <> '' THEN
			MemSet(	destAddr:=ADR(_WriteData.bArray),
					fillByte:=0,
					n:=SIZEOF(_WriteData.bArray));
			MemCpy(	destAddr:=ADR(_WriteData.sString),
					srcAddr:=ADR(_DataToWrite),
					n:=INT_TO_DWORD(LEN(_DataToWrite)));
			_fbTcpWrite.xExecute := TRUE;
		END_IF
	END_IF
	
	_fbTcpWrite(xExecute := _fbTcpWrite.xExecute AND NOT _fbTcpWrite.xDone AND NOT _fbTcpWrite.xError,
				xBusy=>bBusyWrite,
				xDone=>bDoneWrite,
				itfConnection := _fbTcpClient.itfConnection, 
				udiTimeOut := 1000000, // us 
				udiSize := INT_TO_UDINT(LEN(_WriteData.sString)), 
				pData := ADR(_WriteData.bArray));

{endregion}


{region "read"}

	_Read := (_ConnectStep = ConnectStep_CONN);
	CASE _ReadStep OF
			 
		ReadStep_RESET: // RESET
			_fbTcpRead.xEnable := FALSE;
			_ReadStep := ReadStep_IDLE;

		ReadStep_IDLE: // IDLE
			IF _Read THEN
				_ReadStep := ReadStep_ENABLE;
			END_IF

		ReadStep_ENABLE: // ENABLE
			_fbTcpRead.xEnable := TRUE;
			_ReadStep := ReadStep_MONITOR;

